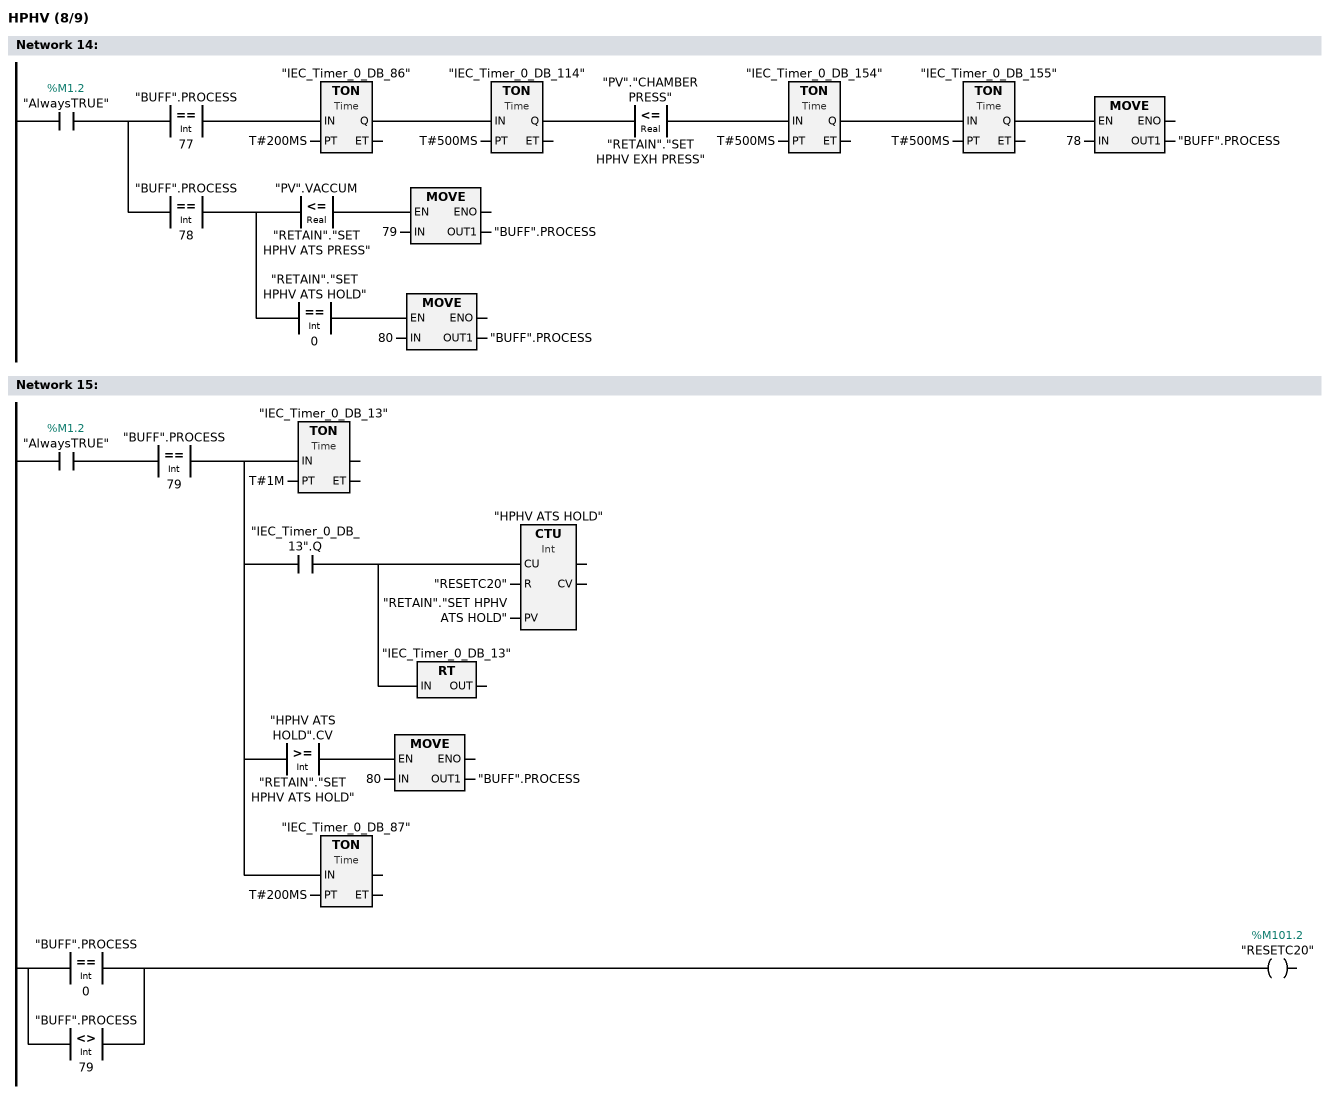
   RUNG wire#powerrail
      Contact( "AlwaysTRUE" )
      wire#w1
      { S7_Templates := "SrcType := Int" } EQ_Contact(in1 := "BUFF".PROCESS, in2 := 77)
      { S7_Templates := "time_type := Time" } "IEC_Timer_0_DB_86".TON(pt := T#200MS, et =>)
      { S7_Templates := "time_type := Time" } "IEC_Timer_0_DB_114".TON(pt := T#500MS, et =>)
      { S7_Templates := "SrcType := Real" } LE_Contact(in1 := "PV"."CHAMBER PRESS", in2 := "RETAIN"."SET HPHV EXH PRESS")
      { S7_Templates := "time_type := Time" } "IEC_Timer_0_DB_154".TON(pt := T#500MS, et =>)
      { S7_Templates := "time_type := Time" } "IEC_Timer_0_DB_155".TON(pt := T#500MS, et =>)
      Move(in := 78, out1 => "BUFF".PROCESS)
   END_RUNG
   RUNG wire#w1
      { S7_Templates := "SrcType := Int" } EQ_Contact(in1 := "BUFF".PROCESS, in2 := 78)
      wire#w2
      { S7_Templates := "SrcType := Real" } LE_Contact(in1 := "PV".VACCUM, in2 := "RETAIN"."SET HPHV ATS PRESS")
      Move(in := 79, out1 => "BUFF".PROCESS)
   END_RUNG
   RUNG wire#w2
      { S7_Templates := "SrcType := Int" } EQ_Contact(in1 := "RETAIN"."SET HPHV ATS HOLD", in2 := 0)
      Move(in := 80, out1 => "BUFF".PROCESS)
   END_RUNG
   // the same network as SCL:
   "IEC_Timer_0_DB_86".TON(IN := "AlwaysTRUE" AND ("BUFF".PROCESS = 77), PT := T#200MS);
   "IEC_Timer_0_DB_114".TON(IN := "IEC_Timer_0_DB_86".Q, PT := T#500MS);
   "IEC_Timer_0_DB_154".TON(IN := "IEC_Timer_0_DB_114".Q AND ("PV"."CHAMBER PRESS" <= "RETAIN"."SET HPHV EXH PRESS"),
                           PT := T#500MS);
   "IEC_Timer_0_DB_155".TON(IN := "IEC_Timer_0_DB_154".Q, PT := T#500MS);
   IF "IEC_Timer_0_DB_155".Q THEN "BUFF".PROCESS := 78; END_IF;
   #_w1 := "AlwaysTRUE" AND ("BUFF".PROCESS = 78);
   IF #_w1 AND ("PV".VACCUM <= "RETAIN"."SET HPHV ATS PRESS") THEN "BUFF".PROCESS := 79; END_IF;
   IF #_w1 AND ("RETAIN"."SET HPHV ATS HOLD" = 0) THEN "BUFF".PROCESS := 80; END_IF;
END_REGION

REGION Network 15
   RUNG wire#powerrail
      Contact( "AlwaysTRUE" )
      { S7_Templates := "SrcType := Int" } EQ_Contact(in1 := "BUFF".PROCESS, in2 := 79)
      wire#w1
      { S7_Templates := "time_type := Time" } "IEC_Timer_0_DB_13".TON(pt := T#1M, et =>)
   END_RUNG
   RUNG wire#w1
      Contact( "IEC_Timer_0_DB_13".Q )
      wire#w2
      { S7_Templates := "value_type := Int" } "HPHV ATS HOLD".CTU(r := "RESETC20", pv := "RETAIN"."SET HPHV ATS HOLD", cv =>)
   END_RUNG
   RUNG wire#w2
      RT_Coil( "IEC_Timer_0_DB_13" )
   END_RUNG
   RUNG wire#w1
      { S7_Templates := "SrcType := Int" } GE_Contact(in1 := "HPHV ATS HOLD".CV, in2 := "RETAIN"."SET HPHV ATS HOLD")
      Move(in := 80, out1 => "BUFF".PROCESS)
   END_RUNG
   RUNG wire#w1
      { S7_Templates := "time_type := Time" } "IEC_Timer_0_DB_87".TON(pt := T#200MS, et =>)
   END_RUNG
   RUNG wire#powerrail
      { S7_Templates := "SrcType := Int" } EQ_Contact(in1 := "BUFF".PROCESS, in2 := 0)
      wire#w3
      Coil( "RESETC20" )
   END_RUNG
   RUNG wire#powerrail
      { S7_Templates := "SrcType := Int" } NE_Contact(in1 := "BUFF".PROCESS, in2 := 79)
   END_RUNG wire#w3
   // the same network as SCL:
   #_w1 := "AlwaysTRUE" AND ("BUFF".PROCESS = 79);
   "IEC_Timer_0_DB_13".TON(IN := #_w1, PT := T#1M);
   #_w2 := #_w1 AND "IEC_Timer_0_DB_13".Q;
   "HPHV ATS HOLD".CTU(CU := #_w2, R := "RESETC20", PV := "RETAIN"."SET HPHV ATS HOLD");
   IF #_w2 THEN RESET_TIMER("IEC_Timer_0_DB_13"); END_IF;
   IF #_w1 AND ("HPHV ATS HOLD".CV >= "RETAIN"."SET HPHV ATS HOLD") THEN "BUFF".PROCESS := 80; END_IF;
   "IEC_Timer_0_DB_87".TON(IN := #_w1, PT := T#200MS);
   "RESETC20" := ("BUFF".PROCESS = 0) OR ("BUFF".PROCESS <> 79);
END_REGION

REGION Network 16
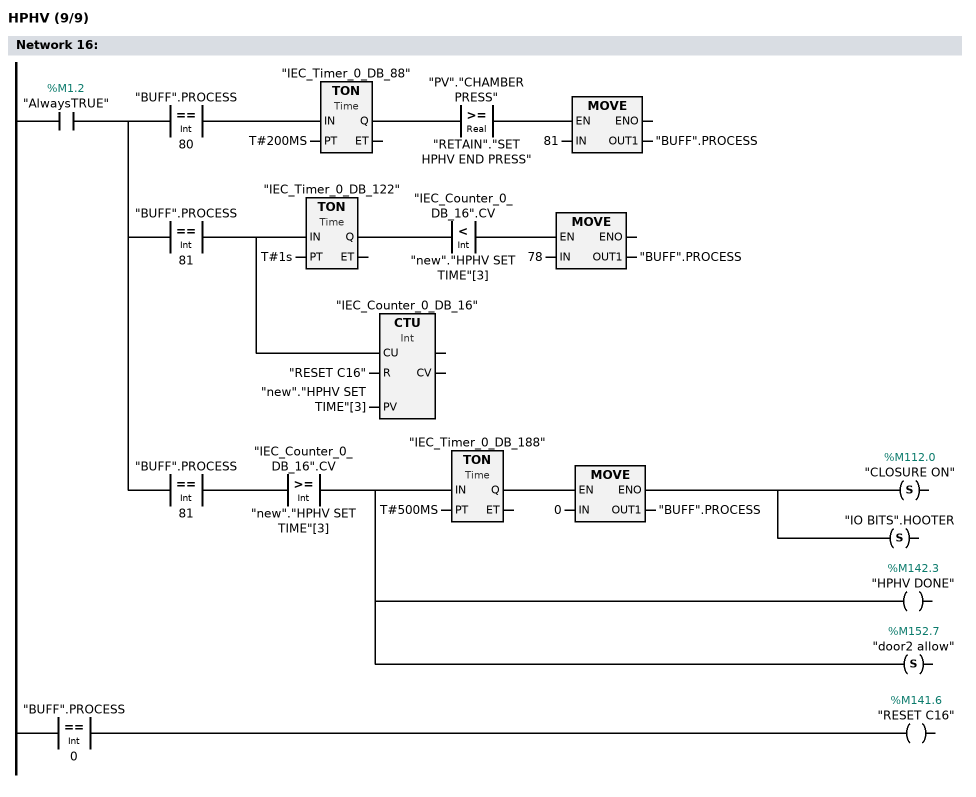
   RUNG wire#powerrail
      Contact( "AlwaysTRUE" )
      wire#w1
      { S7_Templates := "SrcType := Int" } EQ_Contact(in1 := "BUFF".PROCESS, in2 := 80)
      { S7_Templates := "time_type := Time" } "IEC_Timer_0_DB_88".TON(pt := T#200MS, et =>)
      { S7_Templates := "SrcType := Real" } GE_Contact(in1 := "PV"."CHAMBER PRESS", in2 := "RETAIN"."SET HPHV END PRESS")
      Move(in := 81, out1 => "BUFF".PROCESS)
   END_RUNG
   RUNG wire#w1
      { S7_Templates := "SrcType := Int" } EQ_Contact(in1 := "BUFF".PROCESS, in2 := 81)
      wire#w2
      { S7_Templates := "time_type := Time" } "IEC_Timer_0_DB_122".TON(pt := T#1s, et =>)
      { S7_Templates := "SrcType := Int" } LT_Contact(in1 := "IEC_Counter_0_DB_16".CV, in2 := "new"."HPHV SET TIME"[3])
      Move(in := 78, out1 => "BUFF".PROCESS)
   END_RUNG
   RUNG wire#w2
      { S7_Templates := "value_type := Int" } "IEC_Counter_0_DB_16".CTU(r := "RESET C16", pv := "new"."HPHV SET TIME"[3], cv =>)
   END_RUNG
   RUNG wire#w1
      { S7_Templates := "SrcType := Int" } EQ_Contact(in1 := "BUFF".PROCESS, in2 := 81)
      { S7_Templates := "SrcType := Int" } GE_Contact(in1 := "IEC_Counter_0_DB_16".CV, in2 := "new"."HPHV SET TIME"[3])
      wire#w3
      { S7_Templates := "time_type := Time" } "IEC_Timer_0_DB_188".TON(pt := T#500MS, et =>)
      Move(in := 0, out1 => "BUFF".PROCESS)
      wire#w4
      S_Coil( "CLOSURE ON" )
   END_RUNG
   RUNG wire#w4
      S_Coil( "IO BITS".HOOTER )
   END_RUNG
   RUNG wire#w3
      Coil( "HPHV DONE" )
   END_RUNG
   RUNG wire#w3
      S_Coil( "door2 allow" )
   END_RUNG
   RUNG wire#powerrail
      { S7_Templates := "SrcType := Int" } EQ_Contact(in1 := "BUFF".PROCESS, in2 := 0)
      Coil( "RESET C16" )
   END_RUNG
   // the same network as SCL:
   "IEC_Timer_0_DB_88".TON(IN := "AlwaysTRUE" AND ("BUFF".PROCESS = 80), PT := T#200MS);
   IF "IEC_Timer_0_DB_88".Q AND ("PV"."CHAMBER PRESS" >= "RETAIN"."SET HPHV END PRESS") THEN
       "BUFF".PROCESS := 81;
   END_IF;
   #_w1 := "AlwaysTRUE" AND ("BUFF".PROCESS = 81);
   "IEC_Timer_0_DB_122".TON(IN := #_w1, PT := T#1s);
   IF "IEC_Timer_0_DB_122".Q AND ("IEC_Counter_0_DB_16".CV < "new"."HPHV SET TIME"[3]) THEN
       "BUFF".PROCESS := 78;
   END_IF;
   "IEC_Counter_0_DB_16".CTU(CU := #_w1, R := "RESET C16", PV := "new"."HPHV SET TIME"[3]);
   #_w2 := "AlwaysTRUE" AND ("BUFF".PROCESS = 81) AND ("IEC_Counter_0_DB_16".CV >= "new"."HPHV SET TIME"[3]);
   "IEC_Timer_0_DB_188".TON(IN := #_w2, PT := T#500MS);
   IF "IEC_Timer_0_DB_188".Q THEN
       "BUFF".PROCESS := 0;
       "CLOSURE ON" := TRUE;
       "IO BITS".HOOTER := TRUE;
   END_IF;
   "HPHV DONE" := #_w2;
   IF #_w2 THEN "door2 allow" := TRUE; END_IF;
   "RESET C16" := "BUFF".PROCESS = 0;
END_REGION
END_FUNCTION

FUNCTION "BOWIE" : Void   // FC7, LAD
{ S7_Optimized_Access := 'TRUE' }
// stored: SetENOAutomatically false
   VAR_TEMP
      START : Bool;
   END_VAR
   VAR_TEMP   // added for the SCL form of the ladder/FBD networks
      _w1 : Bool;
      _w2 : Bool;
      _w3 : Bool;
      _w4 : Bool;
   END_VAR
BEGIN

REGION Network 1
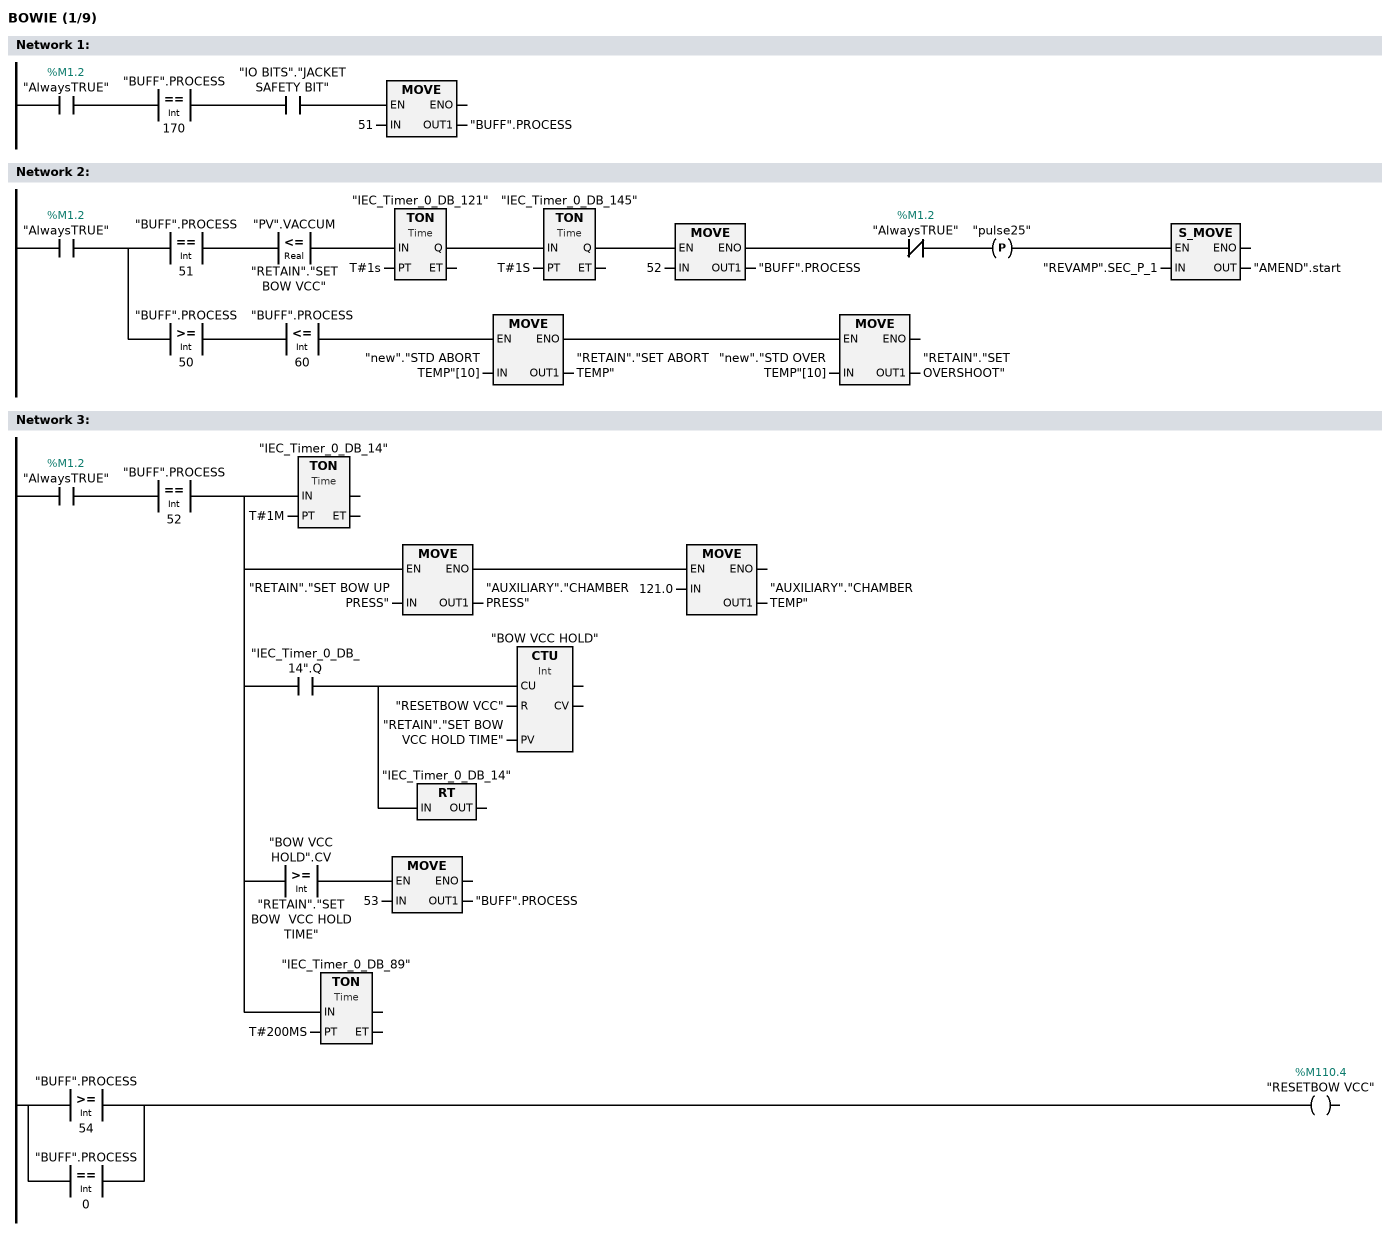
   RUNG wire#powerrail
      Contact( "AlwaysTRUE" )
      { S7_Templates := "SrcType := Int" } EQ_Contact(in1 := "BUFF".PROCESS, in2 := 170)
      Contact( "IO BITS"."JACKET SAFETY BIT" )
      Move(in := 51, out1 => "BUFF".PROCESS)
   END_RUNG
   // the same network as SCL:
   IF "AlwaysTRUE" AND ("BUFF".PROCESS = 170) AND "IO BITS"."JACKET SAFETY BIT" THEN
       "BUFF".PROCESS := 51;
   END_IF;
END_REGION

REGION Network 2
   RUNG wire#powerrail
      Contact( "AlwaysTRUE" )
      wire#w1
      { S7_Templates := "SrcType := Int" } EQ_Contact(in1 := "BUFF".PROCESS, in2 := 51)
      { S7_Templates := "SrcType := Real" } LE_Contact(in1 := "PV".VACCUM, in2 := "RETAIN"."SET BOW VCC")
      { S7_Templates := "time_type := Time" } "IEC_Timer_0_DB_121".TON(pt := T#1s, et =>)
      { S7_Templates := "time_type := Time" } "IEC_Timer_0_DB_145".TON(pt := T#1S, et =>)
      Move(in := 52, out1 => "BUFF".PROCESS)
      I_Contact( "AlwaysTRUE" )
      P_Trig( "pulse25" )
      S_Move(in := "REVAMP".SEC_P_1, out => "AMEND".start)
   END_RUNG
   RUNG wire#w1
      { S7_Templates := "SrcType := Int" } GE_Contact(in1 := "BUFF".PROCESS, in2 := 50)
      { S7_Templates := "SrcType := Int" } LE_Contact(in1 := "BUFF".PROCESS, in2 := 60)
      Move(in := "new"."STD ABORT TEMP"[10], out1 => "RETAIN"."SET ABORT TEMP")
      Move(in := "new"."STD OVER TEMP"[10], out1 => "RETAIN"."SET OVERSHOOT")
   END_RUNG
   // the same network as SCL:
   "IEC_Timer_0_DB_121".TON(IN := "AlwaysTRUE" AND ("BUFF".PROCESS = 51) AND ("PV".VACCUM <= "RETAIN"."SET BOW VCC"),
                           PT := T#1s);
   "IEC_Timer_0_DB_145".TON(IN := "IEC_Timer_0_DB_121".Q, PT := T#1S);
   IF "IEC_Timer_0_DB_145".Q THEN "BUFF".PROCESS := 52; END_IF;
   #_w1 := "IEC_Timer_0_DB_145".Q AND NOT "AlwaysTRUE";
   #_w2 := #_w1 AND NOT "pulse25";   // rising edge
   "pulse25" := #_w1;
   IF #_w2 THEN "AMEND".start := "REVAMP".SEC_P_1; END_IF;
   IF "AlwaysTRUE" AND ("BUFF".PROCESS >= 50) AND ("BUFF".PROCESS <= 60) THEN
       "RETAIN"."SET ABORT TEMP" := "new"."STD ABORT TEMP"[10];
       "RETAIN"."SET OVERSHOOT" := "new"."STD OVER TEMP"[10];
   END_IF;
END_REGION

REGION Network 3
   RUNG wire#powerrail
      Contact( "AlwaysTRUE" )
      { S7_Templates := "SrcType := Int" } EQ_Contact(in1 := "BUFF".PROCESS, in2 := 52)
      wire#w1
      { S7_Templates := "time_type := Time" } "IEC_Timer_0_DB_14".TON(pt := T#1M, et =>)
   END_RUNG
   RUNG wire#w1
      Move(in := "RETAIN"."SET BOW UP PRESS", out1 => "AUXILIARY"."CHAMBER PRESS")
      Move(in := 121.0, out1 => "AUXILIARY"."CHAMBER TEMP")
   END_RUNG
   RUNG wire#w1
      Contact( "IEC_Timer_0_DB_14".Q )
      wire#w2
      { S7_Templates := "value_type := Int" } "BOW VCC HOLD".CTU(r := "RESETBOW VCC", pv := "RETAIN"."SET BOW  VCC HOLD TIME", cv =>)
   END_RUNG
   RUNG wire#w2
      RT_Coil( "IEC_Timer_0_DB_14" )
   END_RUNG
   RUNG wire#w1
      { S7_Templates := "SrcType := Int" } GE_Contact(in1 := "BOW VCC HOLD".CV, in2 := "RETAIN"."SET BOW  VCC HOLD TIME")
      Move(in := 53, out1 => "BUFF".PROCESS)
   END_RUNG
   RUNG wire#w1
      { S7_Templates := "time_type := Time" } "IEC_Timer_0_DB_89".TON(pt := T#200MS, et =>)
   END_RUNG
   RUNG wire#powerrail
      { S7_Templates := "SrcType := Int" } GE_Contact(in1 := "BUFF".PROCESS, in2 := 54)
      wire#w3
      Coil( "RESETBOW VCC" )
   END_RUNG
   RUNG wire#powerrail
      { S7_Templates := "SrcType := Int" } EQ_Contact(in1 := "BUFF".PROCESS, in2 := 0)
   END_RUNG wire#w3
   // the same network as SCL:
   #_w1 := "AlwaysTRUE" AND ("BUFF".PROCESS = 52);
   "IEC_Timer_0_DB_14".TON(IN := #_w1, PT := T#1M);
   IF #_w1 THEN
       "AUXILIARY"."CHAMBER PRESS" := "RETAIN"."SET BOW UP PRESS";
       "AUXILIARY"."CHAMBER TEMP" := 121.0;
   END_IF;
   #_w2 := #_w1 AND "IEC_Timer_0_DB_14".Q;
   "BOW VCC HOLD".CTU(CU := #_w2, R := "RESETBOW VCC", PV := "RETAIN"."SET BOW  VCC HOLD TIME");
   IF #_w2 THEN RESET_TIMER("IEC_Timer_0_DB_14"); END_IF;
   IF #_w1 AND ("BOW VCC HOLD".CV >= "RETAIN"."SET BOW  VCC HOLD TIME") THEN "BUFF".PROCESS := 53; END_IF;
   "IEC_Timer_0_DB_89".TON(IN := #_w1, PT := T#200MS);
   "RESETBOW VCC" := ("BUFF".PROCESS >= 54) OR ("BUFF".PROCESS = 0);
END_REGION

REGION Network 4
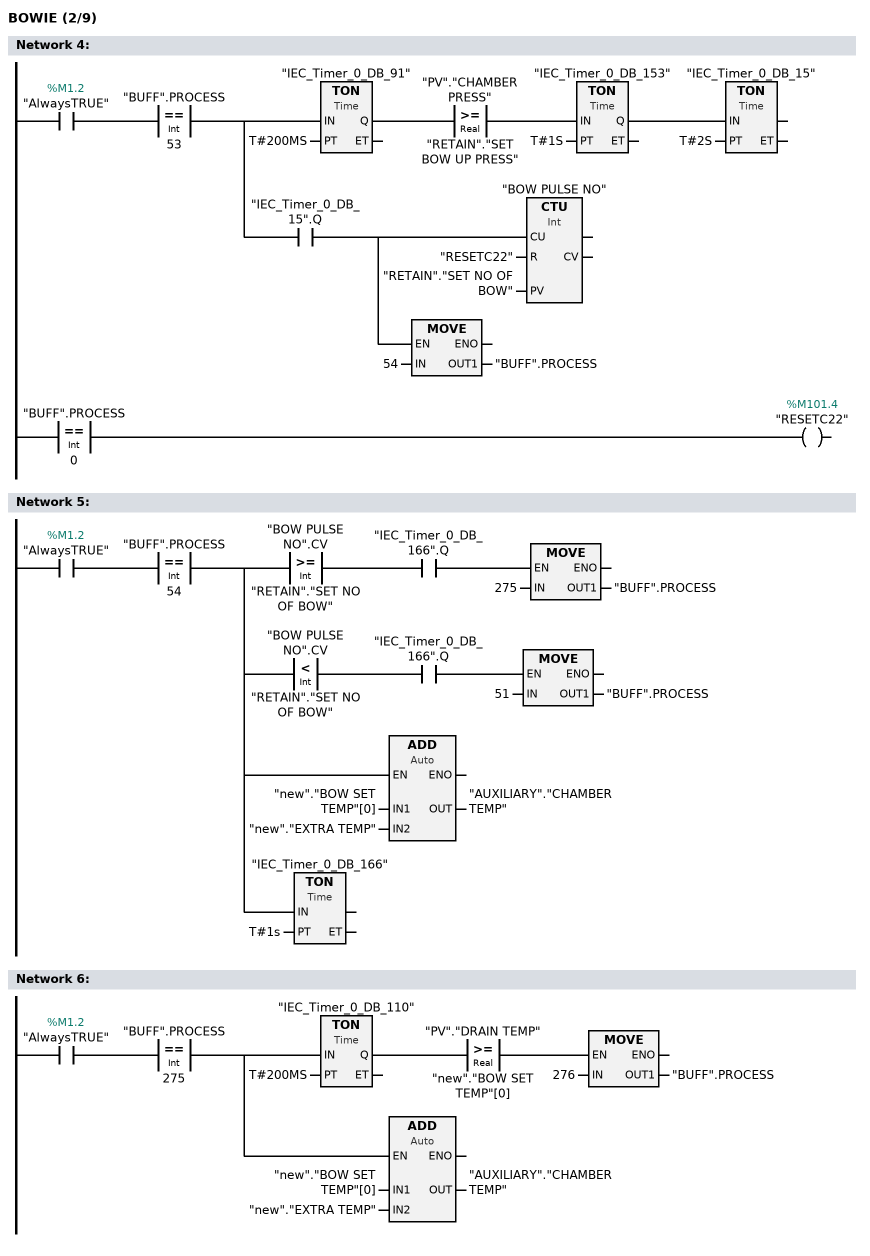
   RUNG wire#powerrail
      Contact( "AlwaysTRUE" )
      { S7_Templates := "SrcType := Int" } EQ_Contact(in1 := "BUFF".PROCESS, in2 := 53)
      wire#w1
      { S7_Templates := "time_type := Time" } "IEC_Timer_0_DB_91".TON(pt := T#200MS, et =>)
      { S7_Templates := "SrcType := Real" } GE_Contact(in1 := "PV"."CHAMBER PRESS", in2 := "RETAIN"."SET BOW UP PRESS")
      { S7_Templates := "time_type := Time" } "IEC_Timer_0_DB_153".TON(pt := T#1S, et =>)
      { S7_Templates := "time_type := Time" } "IEC_Timer_0_DB_15".TON(pt := T#2S, et =>)
   END_RUNG
   RUNG wire#w1
      Contact( "IEC_Timer_0_DB_15".Q )
      wire#w2
      { S7_Templates := "value_type := Int" } "BOW PULSE NO".CTU(r := "RESETC22", pv := "RETAIN"."SET NO OF BOW", cv =>)
   END_RUNG
   RUNG wire#w2
      Move(in := 54, out1 => "BUFF".PROCESS)
   END_RUNG
   RUNG wire#powerrail
      { S7_Templates := "SrcType := Int" } EQ_Contact(in1 := "BUFF".PROCESS, in2 := 0)
      Coil( "RESETC22" )
   END_RUNG
   // the same network as SCL:
   #_w1 := "AlwaysTRUE" AND ("BUFF".PROCESS = 53);
   "IEC_Timer_0_DB_91".TON(IN := #_w1, PT := T#200MS);
   "IEC_Timer_0_DB_153".TON(IN := "IEC_Timer_0_DB_91".Q AND ("PV"."CHAMBER PRESS" >= "RETAIN"."SET BOW UP PRESS"),
                           PT := T#1S);
   "IEC_Timer_0_DB_15".TON(IN := "IEC_Timer_0_DB_153".Q, PT := T#2S);
   #_w2 := #_w1 AND "IEC_Timer_0_DB_15".Q;
   "BOW PULSE NO".CTU(CU := #_w2, R := "RESETC22", PV := "RETAIN"."SET NO OF BOW");
   IF #_w2 THEN "BUFF".PROCESS := 54; END_IF;
   "RESETC22" := "BUFF".PROCESS = 0;
END_REGION

REGION Network 5
   RUNG wire#powerrail
      Contact( "AlwaysTRUE" )
      { S7_Templates := "SrcType := Int" } EQ_Contact(in1 := "BUFF".PROCESS, in2 := 54)
      wire#w1
      { S7_Templates := "SrcType := Int" } GE_Contact(in1 := "BOW PULSE NO".CV, in2 := "RETAIN"."SET NO OF BOW")
      Contact( "IEC_Timer_0_DB_166".Q )
      Move(in := 275, out1 => "BUFF".PROCESS)
   END_RUNG
   RUNG wire#w1
      { S7_Templates := "SrcType := Int" } LT_Contact(in1 := "BOW PULSE NO".CV, in2 := "RETAIN"."SET NO OF BOW")
      Contact( "IEC_Timer_0_DB_166".Q )
      Move(in := 51, out1 => "BUFF".PROCESS)
   END_RUNG
   RUNG wire#w1
      Add(in1 := "new"."BOW SET TEMP"[0], in2 := "new"."EXTRA TEMP", out => "AUXILIARY"."CHAMBER TEMP")
   END_RUNG
   RUNG wire#w1
      { S7_Templates := "time_type := Time" } "IEC_Timer_0_DB_166".TON(pt := T#1s, et =>)
   END_RUNG
   // the same network as SCL:
   #_w1 := "AlwaysTRUE" AND ("BUFF".PROCESS = 54);
   IF #_w1 AND ("BOW PULSE NO".CV >= "RETAIN"."SET NO OF BOW") AND "IEC_Timer_0_DB_166".Q THEN
       "BUFF".PROCESS := 275;
   END_IF;
   IF #_w1 AND ("BOW PULSE NO".CV < "RETAIN"."SET NO OF BOW") AND "IEC_Timer_0_DB_166".Q THEN
       "BUFF".PROCESS := 51;
   END_IF;
   IF #_w1 THEN "AUXILIARY"."CHAMBER TEMP" := "new"."BOW SET TEMP"[0] + "new"."EXTRA TEMP"; END_IF;
   "IEC_Timer_0_DB_166".TON(IN := #_w1, PT := T#1s);
END_REGION

REGION Network 6
   RUNG wire#powerrail
      Contact( "AlwaysTRUE" )
      { S7_Templates := "SrcType := Int" } EQ_Contact(in1 := "BUFF".PROCESS, in2 := 275)
      wire#w1
      { S7_Templates := "time_type := Time" } "IEC_Timer_0_DB_110".TON(pt := T#200MS, et =>)
      { S7_Templates := "SrcType := Real" } GE_Contact(in1 := "PV"."DRAIN TEMP", in2 := "new"."BOW SET TEMP"[0])
      Move(in := 276, out1 => "BUFF".PROCESS)
   END_RUNG
   RUNG wire#w1
      Add(in1 := "new"."BOW SET TEMP"[0], in2 := "new"."EXTRA TEMP", out => "AUXILIARY"."CHAMBER TEMP")
   END_RUNG
   // the same network as SCL:
   #_w1 := "AlwaysTRUE" AND ("BUFF".PROCESS = 275);
   "IEC_Timer_0_DB_110".TON(IN := #_w1, PT := T#200MS);
   IF "IEC_Timer_0_DB_110".Q AND ("PV"."DRAIN TEMP" >= "new"."BOW SET TEMP"[0]) THEN
       "BUFF".PROCESS := 276;
   END_IF;
   IF #_w1 THEN "AUXILIARY"."CHAMBER TEMP" := "new"."BOW SET TEMP"[0] + "new"."EXTRA TEMP"; END_IF;
END_REGION

REGION Network 7
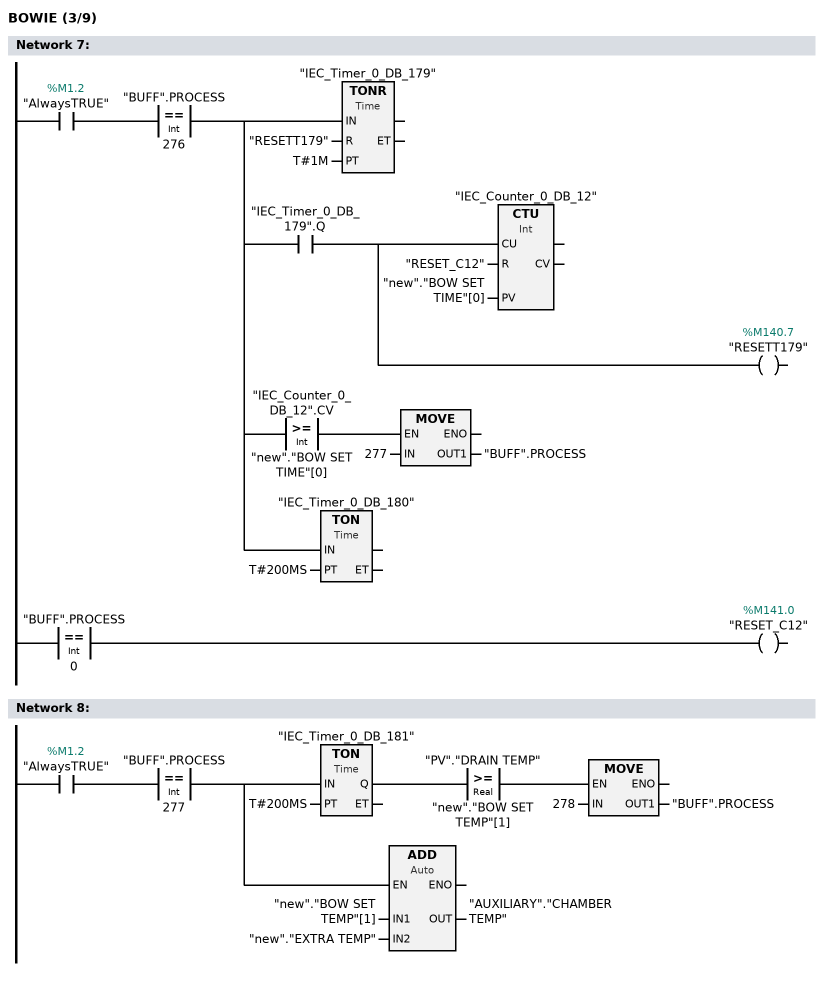
   RUNG wire#powerrail
      Contact( "AlwaysTRUE" )
      { S7_Templates := "SrcType := Int" } EQ_Contact(in1 := "BUFF".PROCESS, in2 := 276)
      wire#w1
      { S7_Templates := "time_type := Time" } "IEC_Timer_0_DB_179".TONR(r := "RESETT179", pt := T#1M, et =>)
   END_RUNG
   RUNG wire#w1
      Contact( "IEC_Timer_0_DB_179".Q )
      wire#w2
      { S7_Templates := "value_type := Int" } "IEC_Counter_0_DB_12".CTU(r := "RESET_C12", pv := "new"."BOW SET TIME"[0], cv =>)
   END_RUNG
   RUNG wire#w2
      Coil( "RESETT179" )
   END_RUNG
   RUNG wire#w1
      { S7_Templates := "SrcType := Int" } GE_Contact(in1 := "IEC_Counter_0_DB_12".CV, in2 := "new"."BOW SET TIME"[0])
      Move(in := 277, out1 => "BUFF".PROCESS)
   END_RUNG
   RUNG wire#w1
      { S7_Templates := "time_type := Time" } "IEC_Timer_0_DB_180".TON(pt := T#200MS, et =>)
   END_RUNG
   RUNG wire#powerrail
      { S7_Templates := "SrcType := Int" } EQ_Contact(in1 := "BUFF".PROCESS, in2 := 0)
      Coil( "RESET_C12" )
   END_RUNG
   // the same network as SCL:
   #_w1 := "AlwaysTRUE" AND ("BUFF".PROCESS = 276);
   "IEC_Timer_0_DB_179".TONR(IN := #_w1, R := "RESETT179", PT := T#1M);
   #_w2 := #_w1 AND "IEC_Timer_0_DB_179".Q;
   "IEC_Counter_0_DB_12".CTU(CU := #_w2, R := "RESET_C12", PV := "new"."BOW SET TIME"[0]);
   "RESETT179" := #_w2;
   IF #_w1 AND ("IEC_Counter_0_DB_12".CV >= "new"."BOW SET TIME"[0]) THEN "BUFF".PROCESS := 277; END_IF;
   "IEC_Timer_0_DB_180".TON(IN := #_w1, PT := T#200MS);
   "RESET_C12" := "BUFF".PROCESS = 0;
END_REGION

REGION Network 8
   RUNG wire#powerrail
      Contact( "AlwaysTRUE" )
      { S7_Templates := "SrcType := Int" } EQ_Contact(in1 := "BUFF".PROCESS, in2 := 277)
      wire#w1
      { S7_Templates := "time_type := Time" } "IEC_Timer_0_DB_181".TON(pt := T#200MS, et =>)
      { S7_Templates := "SrcType := Real" } GE_Contact(in1 := "PV"."DRAIN TEMP", in2 := "new"."BOW SET TEMP"[1])
      Move(in := 278, out1 => "BUFF".PROCESS)
   END_RUNG
   RUNG wire#w1
      Add(in1 := "new"."BOW SET TEMP"[1], in2 := "new"."EXTRA TEMP", out => "AUXILIARY"."CHAMBER TEMP")
   END_RUNG
   // the same network as SCL:
   #_w1 := "AlwaysTRUE" AND ("BUFF".PROCESS = 277);
   "IEC_Timer_0_DB_181".TON(IN := #_w1, PT := T#200MS);
   IF "IEC_Timer_0_DB_181".Q AND ("PV"."DRAIN TEMP" >= "new"."BOW SET TEMP"[1]) THEN
       "BUFF".PROCESS := 278;
   END_IF;
   IF #_w1 THEN "AUXILIARY"."CHAMBER TEMP" := "new"."BOW SET TEMP"[1] + "new"."EXTRA TEMP"; END_IF;
END_REGION

REGION Network 9
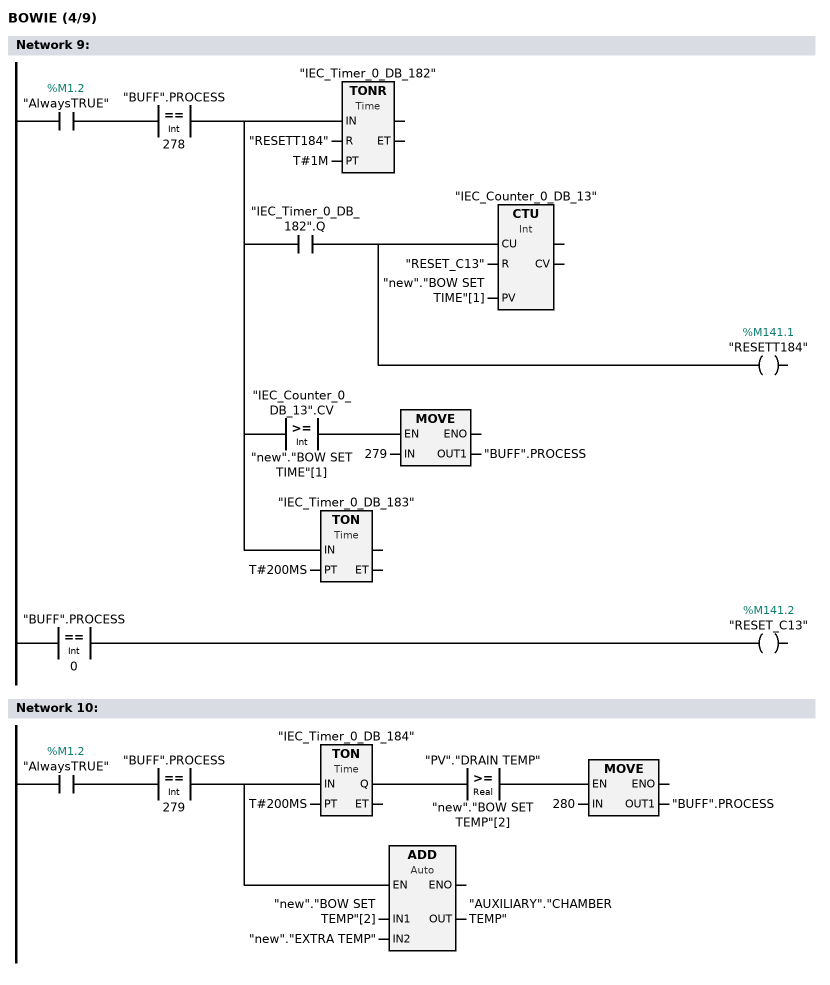
   RUNG wire#powerrail
      Contact( "AlwaysTRUE" )
      { S7_Templates := "SrcType := Int" } EQ_Contact(in1 := "BUFF".PROCESS, in2 := 278)
      wire#w1
      { S7_Templates := "time_type := Time" } "IEC_Timer_0_DB_182".TONR(r := "RESETT184", pt := T#1M, et =>)
   END_RUNG
   RUNG wire#w1
      Contact( "IEC_Timer_0_DB_182".Q )
      wire#w2
      { S7_Templates := "value_type := Int" } "IEC_Counter_0_DB_13".CTU(r := "RESET_C13", pv := "new"."BOW SET TIME"[1], cv =>)
   END_RUNG
   RUNG wire#w2
      Coil( "RESETT184" )
   END_RUNG
   RUNG wire#w1
      { S7_Templates := "SrcType := Int" } GE_Contact(in1 := "IEC_Counter_0_DB_13".CV, in2 := "new"."BOW SET TIME"[1])
      Move(in := 279, out1 => "BUFF".PROCESS)
   END_RUNG
   RUNG wire#w1
      { S7_Templates := "time_type := Time" } "IEC_Timer_0_DB_183".TON(pt := T#200MS, et =>)
   END_RUNG
   RUNG wire#powerrail
      { S7_Templates := "SrcType := Int" } EQ_Contact(in1 := "BUFF".PROCESS, in2 := 0)
      Coil( "RESET_C13" )
   END_RUNG
   // the same network as SCL:
   #_w1 := "AlwaysTRUE" AND ("BUFF".PROCESS = 278);
   "IEC_Timer_0_DB_182".TONR(IN := #_w1, R := "RESETT184", PT := T#1M);
   #_w2 := #_w1 AND "IEC_Timer_0_DB_182".Q;
   "IEC_Counter_0_DB_13".CTU(CU := #_w2, R := "RESET_C13", PV := "new"."BOW SET TIME"[1]);
   "RESETT184" := #_w2;
   IF #_w1 AND ("IEC_Counter_0_DB_13".CV >= "new"."BOW SET TIME"[1]) THEN "BUFF".PROCESS := 279; END_IF;
   "IEC_Timer_0_DB_183".TON(IN := #_w1, PT := T#200MS);
   "RESET_C13" := "BUFF".PROCESS = 0;
END_REGION

REGION Network 10
   RUNG wire#powerrail
      Contact( "AlwaysTRUE" )
      { S7_Templates := "SrcType := Int" } EQ_Contact(in1 := "BUFF".PROCESS, in2 := 279)
      wire#w1
      { S7_Templates := "time_type := Time" } "IEC_Timer_0_DB_184".TON(pt := T#200MS, et =>)
      { S7_Templates := "SrcType := Real" } GE_Contact(in1 := "PV"."DRAIN TEMP", in2 := "new"."BOW SET TEMP"[2])
      Move(in := 280, out1 => "BUFF".PROCESS)
   END_RUNG
   RUNG wire#w1
      Add(in1 := "new"."BOW SET TEMP"[2], in2 := "new"."EXTRA TEMP", out => "AUXILIARY"."CHAMBER TEMP")
   END_RUNG
   // the same network as SCL:
   #_w1 := "AlwaysTRUE" AND ("BUFF".PROCESS = 279);
   "IEC_Timer_0_DB_184".TON(IN := #_w1, PT := T#200MS);
   IF "IEC_Timer_0_DB_184".Q AND ("PV"."DRAIN TEMP" >= "new"."BOW SET TEMP"[2]) THEN
       "BUFF".PROCESS := 280;
   END_IF;
   IF #_w1 THEN "AUXILIARY"."CHAMBER TEMP" := "new"."BOW SET TEMP"[2] + "new"."EXTRA TEMP"; END_IF;
END_REGION

REGION Network 11
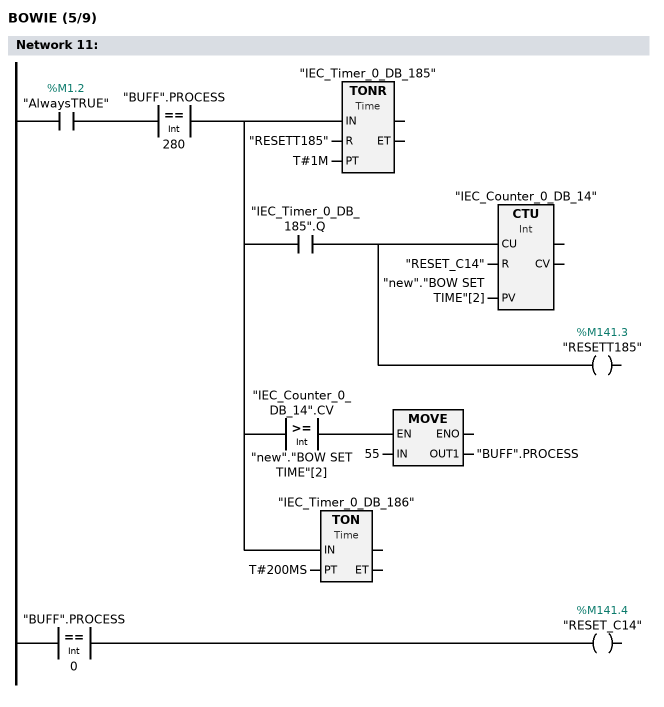
   RUNG wire#powerrail
      Contact( "AlwaysTRUE" )
      { S7_Templates := "SrcType := Int" } EQ_Contact(in1 := "BUFF".PROCESS, in2 := 280)
      wire#w1
      { S7_Templates := "time_type := Time" } "IEC_Timer_0_DB_185".TONR(r := "RESETT185", pt := T#1M, et =>)
   END_RUNG
   RUNG wire#w1
      Contact( "IEC_Timer_0_DB_185".Q )
      wire#w2
      { S7_Templates := "value_type := Int" } "IEC_Counter_0_DB_14".CTU(r := "RESET_C14", pv := "new"."BOW SET TIME"[2], cv =>)
   END_RUNG
   RUNG wire#w2
      Coil( "RESETT185" )
   END_RUNG
   RUNG wire#w1
      { S7_Templates := "SrcType := Int" } GE_Contact(in1 := "IEC_Counter_0_DB_14".CV, in2 := "new"."BOW SET TIME"[2])
      Move(in := 55, out1 => "BUFF".PROCESS)
   END_RUNG
   RUNG wire#w1
      { S7_Templates := "time_type := Time" } "IEC_Timer_0_DB_186".TON(pt := T#200MS, et =>)
   END_RUNG
   RUNG wire#powerrail
      { S7_Templates := "SrcType := Int" } EQ_Contact(in1 := "BUFF".PROCESS, in2 := 0)
      Coil( "RESET_C14" )
   END_RUNG
   // the same network as SCL:
   #_w1 := "AlwaysTRUE" AND ("BUFF".PROCESS = 280);
   "IEC_Timer_0_DB_185".TONR(IN := #_w1, R := "RESETT185", PT := T#1M);
   #_w2 := #_w1 AND "IEC_Timer_0_DB_185".Q;
   "IEC_Counter_0_DB_14".CTU(CU := #_w2, R := "RESET_C14", PV := "new"."BOW SET TIME"[2]);
   "RESETT185" := #_w2;
   IF #_w1 AND ("IEC_Counter_0_DB_14".CV >= "new"."BOW SET TIME"[2]) THEN "BUFF".PROCESS := 55; END_IF;
   "IEC_Timer_0_DB_186".TON(IN := #_w1, PT := T#200MS);
   "RESET_C14" := "BUFF".PROCESS = 0;
END_REGION

REGION Network 12
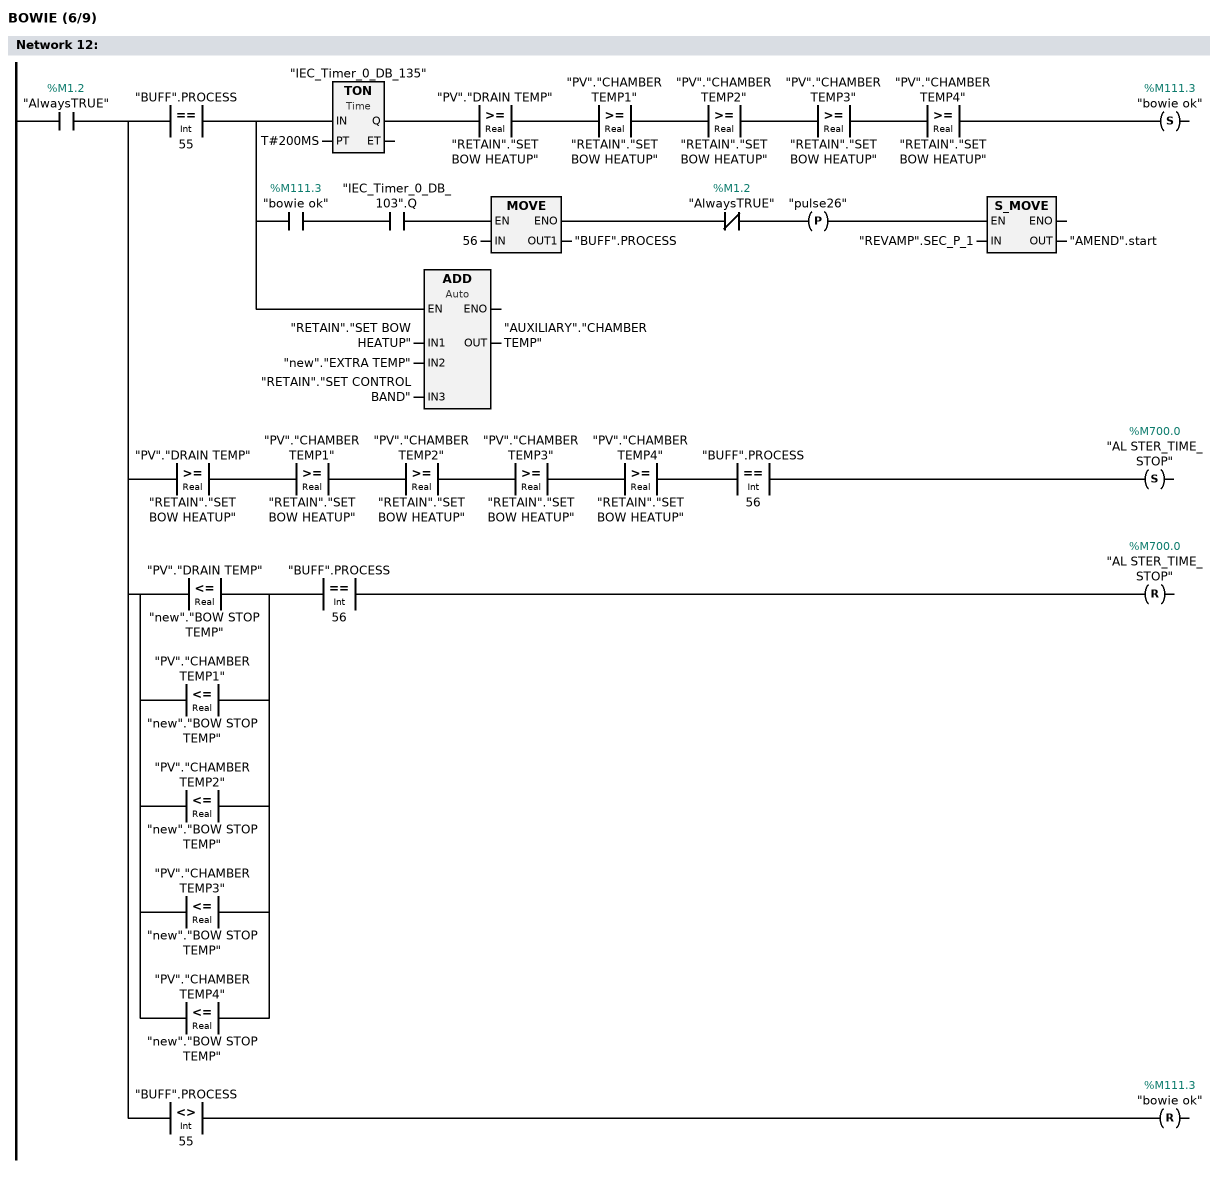
   RUNG wire#powerrail
      Contact( "AlwaysTRUE" )
      wire#w1
      { S7_Templates := "SrcType := Int" } EQ_Contact(in1 := "BUFF".PROCESS, in2 := 55)
      wire#w2
      { S7_Templates := "time_type := Time" } "IEC_Timer_0_DB_135".TON(pt := T#200MS, et =>)
      { S7_Templates := "SrcType := Real" } GE_Contact(in1 := "PV"."DRAIN TEMP", in2 := "RETAIN"."SET BOW HEATUP")
      { S7_Templates := "SrcType := Real" } GE_Contact(in1 := "PV"."CHAMBER TEMP1", in2 := "RETAIN"."SET BOW HEATUP")
      { S7_Templates := "SrcType := Real" } GE_Contact(in1 := "PV"."CHAMBER TEMP2", in2 := "RETAIN"."SET BOW HEATUP")
      { S7_Templates := "SrcType := Real" } GE_Contact(in1 := "PV"."CHAMBER TEMP3", in2 := "RETAIN"."SET BOW HEATUP")
      { S7_Templates := "SrcType := Real" } GE_Contact(in1 := "PV"."CHAMBER TEMP4", in2 := "RETAIN"."SET BOW HEATUP")
      S_Coil( "bowie ok" )
   END_RUNG
   RUNG wire#w2
      Contact( "bowie ok" )
      Contact( "IEC_Timer_0_DB_103".Q )
      Move(in := 56, out1 => "BUFF".PROCESS)
      I_Contact( "AlwaysTRUE" )
      P_Trig( "pulse26" )
      S_Move(in := "REVAMP".SEC_P_1, out => "AMEND".start)
   END_RUNG
   RUNG wire#w2
      Add(in1 := "RETAIN"."SET BOW HEATUP", in2 := "new"."EXTRA TEMP", in3 := "RETAIN"."SET CONTROL BAND", out => "AUXILIARY"."CHAMBER TEMP")
   END_RUNG
   RUNG wire#w1
      { S7_Templates := "SrcType := Real" } GE_Contact(in1 := "PV"."DRAIN TEMP", in2 := "RETAIN"."SET BOW HEATUP")
      { S7_Templates := "SrcType := Real" } GE_Contact(in1 := "PV"."CHAMBER TEMP1", in2 := "RETAIN"."SET BOW HEATUP")
      { S7_Templates := "SrcType := Real" } GE_Contact(in1 := "PV"."CHAMBER TEMP2", in2 := "RETAIN"."SET BOW HEATUP")
      { S7_Templates := "SrcType := Real" } GE_Contact(in1 := "PV"."CHAMBER TEMP3", in2 := "RETAIN"."SET BOW HEATUP")
      { S7_Templates := "SrcType := Real" } GE_Contact(in1 := "PV"."CHAMBER TEMP4", in2 := "RETAIN"."SET BOW HEATUP")
      { S7_Templates := "SrcType := Int" } EQ_Contact(in1 := "BUFF".PROCESS, in2 := 56)
      S_Coil( "AL STER_TIME_STOP" )
   END_RUNG
   RUNG wire#w1
      { S7_Templates := "SrcType := Real" } LE_Contact(in1 := "PV"."DRAIN TEMP", in2 := "new"."BOW STOP TEMP")
      wire#w3
      { S7_Templates := "SrcType := Int" } EQ_Contact(in1 := "BUFF".PROCESS, in2 := 56)
      R_Coil( "AL STER_TIME_STOP" )
   END_RUNG
   RUNG wire#w1
      { S7_Templates := "SrcType := Real" } LE_Contact(in1 := "PV"."CHAMBER TEMP1", in2 := "new"."BOW STOP TEMP")
   END_RUNG wire#w3
   RUNG wire#w1
      { S7_Templates := "SrcType := Real" } LE_Contact(in1 := "PV"."CHAMBER TEMP2", in2 := "new"."BOW STOP TEMP")
   END_RUNG wire#w3
   RUNG wire#w1
      { S7_Templates := "SrcType := Real" } LE_Contact(in1 := "PV"."CHAMBER TEMP3", in2 := "new"."BOW STOP TEMP")
   END_RUNG wire#w3
   RUNG wire#w1
      { S7_Templates := "SrcType := Real" } LE_Contact(in1 := "PV"."CHAMBER TEMP4", in2 := "new"."BOW STOP TEMP")
   END_RUNG wire#w3
   RUNG wire#w1
      { S7_Templates := "SrcType := Int" } NE_Contact(in1 := "BUFF".PROCESS, in2 := 55)
      R_Coil( "bowie ok" )
   END_RUNG
   // the same network as SCL:
   #_w1 := "AlwaysTRUE" AND ("BUFF".PROCESS = 55);
   "IEC_Timer_0_DB_135".TON(IN := #_w1, PT := T#200MS);
   IF "IEC_Timer_0_DB_135".Q AND ("PV"."DRAIN TEMP" >= "RETAIN"."SET BOW HEATUP") AND ("PV"."CHAMBER TEMP1" >= "RETAIN"."SET BOW HEATUP") AND ("PV"."CHAMBER TEMP2" >= "RETAIN"."SET BOW HEATUP") AND ("PV"."CHAMBER TEMP3" >= "RETAIN"."SET BOW HEATUP") AND ("PV"."CHAMBER TEMP4" >= "RETAIN"."SET BOW HEATUP") THEN
       "bowie ok" := TRUE;
   END_IF;
   #_w2 := #_w1 AND "bowie ok" AND "IEC_Timer_0_DB_103".Q;
   IF #_w2 THEN "BUFF".PROCESS := 56; END_IF;
   #_w3 := #_w2 AND NOT "AlwaysTRUE";
   #_w4 := #_w3 AND NOT "pulse26";   // rising edge
   "pulse26" := #_w3;
   IF #_w4 THEN "AMEND".start := "REVAMP".SEC_P_1; END_IF;
   IF #_w1 THEN
       "AUXILIARY"."CHAMBER TEMP" := "RETAIN"."SET BOW HEATUP" + "new"."EXTRA TEMP" + "RETAIN"."SET CONTROL BAND";
   END_IF;
   IF "AlwaysTRUE" AND ("PV"."DRAIN TEMP" >= "RETAIN"."SET BOW HEATUP") AND ("PV"."CHAMBER TEMP1" >= "RETAIN"."SET BOW HEATUP") AND ("PV"."CHAMBER TEMP2" >= "RETAIN"."SET BOW HEATUP") AND ("PV"."CHAMBER TEMP3" >= "RETAIN"."SET BOW HEATUP") AND ("PV"."CHAMBER TEMP4" >= "RETAIN"."SET BOW HEATUP") AND ("BUFF".PROCESS = 56) THEN
       "AL STER_TIME_STOP" := TRUE;
   END_IF;
   IF "AlwaysTRUE" AND (("PV"."DRAIN TEMP" <= "new"."BOW STOP TEMP") OR ("PV"."CHAMBER TEMP1" <= "new"."BOW STOP TEMP") OR ("PV"."CHAMBER TEMP2" <= "new"."BOW STOP TEMP") OR ("PV"."CHAMBER TEMP3" <= "new"."BOW STOP TEMP") OR ("PV"."CHAMBER TEMP4" <= "new"."BOW STOP TEMP")) AND ("BUFF".PROCESS = 56) THEN
       "AL STER_TIME_STOP" := FALSE;
   END_IF;
   IF "AlwaysTRUE" AND ("BUFF".PROCESS <> 55) THEN "bowie ok" := FALSE; END_IF;
END_REGION

REGION Network 13
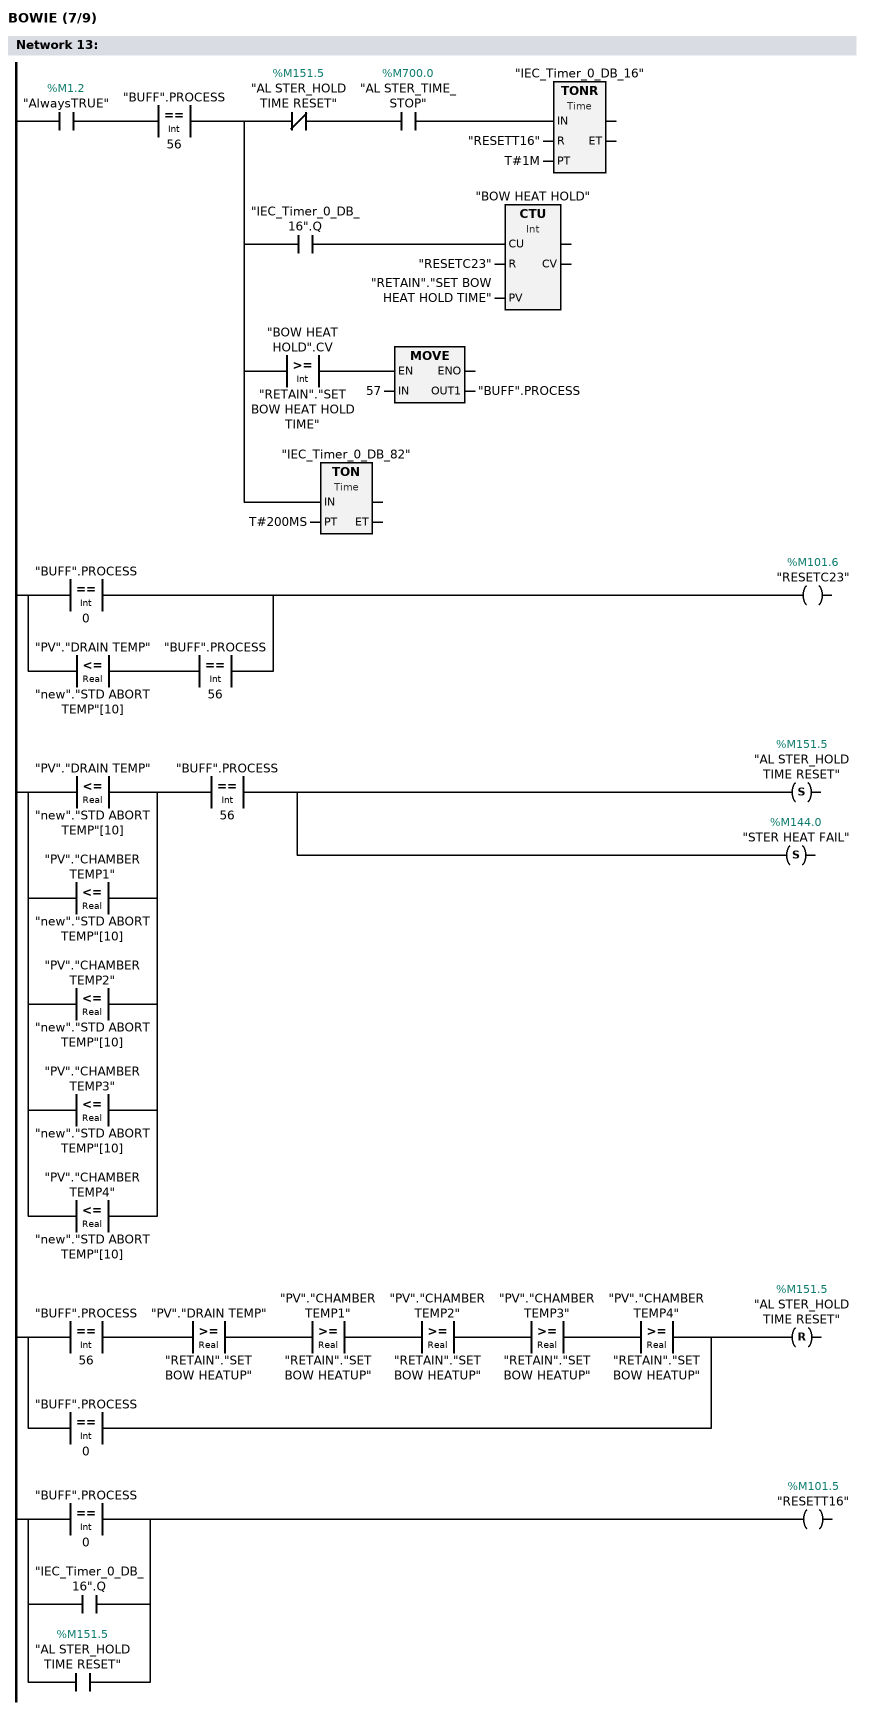
   RUNG wire#powerrail
      Contact( "AlwaysTRUE" )
      { S7_Templates := "SrcType := Int" } EQ_Contact(in1 := "BUFF".PROCESS, in2 := 56)
      wire#w1
      I_Contact( "AL STER_HOLD TIME RESET" )
      Contact( "AL STER_TIME_STOP" )
      { S7_Templates := "time_type := Time" } "IEC_Timer_0_DB_16".TONR(r := "RESETT16", pt := T#1M, et =>)
   END_RUNG
   RUNG wire#w1
      Contact( "IEC_Timer_0_DB_16".Q )
      { S7_Templates := "value_type := Int" } "BOW HEAT HOLD".CTU(r := "RESETC23", pv := "RETAIN"."SET BOW HEAT HOLD TIME", cv =>)
   END_RUNG
   RUNG wire#w1
      { S7_Templates := "SrcType := Int" } GE_Contact(in1 := "BOW HEAT HOLD".CV, in2 := "RETAIN"."SET BOW HEAT HOLD TIME")
      Move(in := 57, out1 => "BUFF".PROCESS)
   END_RUNG
   RUNG wire#w1
      { S7_Templates := "time_type := Time" } "IEC_Timer_0_DB_82".TON(pt := T#200MS, et =>)
   END_RUNG
   RUNG wire#powerrail
      { S7_Templates := "SrcType := Int" } EQ_Contact(in1 := "BUFF".PROCESS, in2 := 0)
      wire#w2
      Coil( "RESETC23" )
   END_RUNG
   RUNG wire#powerrail
      { S7_Templates := "SrcType := Real" } LE_Contact(in1 := "PV"."DRAIN TEMP", in2 := "new"."STD ABORT TEMP"[10])
      { S7_Templates := "SrcType := Int" } EQ_Contact(in1 := "BUFF".PROCESS, in2 := 56)
   END_RUNG wire#w2
   RUNG wire#powerrail
      { S7_Templates := "SrcType := Real" } LE_Contact(in1 := "PV"."DRAIN TEMP", in2 := "new"."STD ABORT TEMP"[10])
      wire#w3
      { S7_Templates := "SrcType := Int" } EQ_Contact(in1 := "BUFF".PROCESS, in2 := 56)
      wire#w4
      S_Coil( "AL STER_HOLD TIME RESET" )
   END_RUNG
   RUNG wire#powerrail
      { S7_Templates := "SrcType := Real" } LE_Contact(in1 := "PV"."CHAMBER TEMP1", in2 := "new"."STD ABORT TEMP"[10])
   END_RUNG wire#w3
   RUNG wire#powerrail
      { S7_Templates := "SrcType := Real" } LE_Contact(in1 := "PV"."CHAMBER TEMP2", in2 := "new"."STD ABORT TEMP"[10])
   END_RUNG wire#w3
   RUNG wire#powerrail
      { S7_Templates := "SrcType := Real" } LE_Contact(in1 := "PV"."CHAMBER TEMP3", in2 := "new"."STD ABORT TEMP"[10])
   END_RUNG wire#w3
   RUNG wire#powerrail
      { S7_Templates := "SrcType := Real" } LE_Contact(in1 := "PV"."CHAMBER TEMP4", in2 := "new"."STD ABORT TEMP"[10])
   END_RUNG wire#w3
   RUNG wire#w4
      S_Coil( "STER HEAT FAIL" )
   END_RUNG
   RUNG wire#powerrail
      { S7_Templates := "SrcType := Int" } EQ_Contact(in1 := "BUFF".PROCESS, in2 := 56)
      { S7_Templates := "SrcType := Real" } GE_Contact(in1 := "PV"."DRAIN TEMP", in2 := "RETAIN"."SET BOW HEATUP")
      { S7_Templates := "SrcType := Real" } GE_Contact(in1 := "PV"."CHAMBER TEMP1", in2 := "RETAIN"."SET BOW HEATUP")
      { S7_Templates := "SrcType := Real" } GE_Contact(in1 := "PV"."CHAMBER TEMP2", in2 := "RETAIN"."SET BOW HEATUP")
      { S7_Templates := "SrcType := Real" } GE_Contact(in1 := "PV"."CHAMBER TEMP3", in2 := "RETAIN"."SET BOW HEATUP")
      { S7_Templates := "SrcType := Real" } GE_Contact(in1 := "PV"."CHAMBER TEMP4", in2 := "RETAIN"."SET BOW HEATUP")
      wire#w5
      R_Coil( "AL STER_HOLD TIME RESET" )
   END_RUNG
   RUNG wire#powerrail
      { S7_Templates := "SrcType := Int" } EQ_Contact(in1 := "BUFF".PROCESS, in2 := 0)
   END_RUNG wire#w5
   RUNG wire#powerrail
      { S7_Templates := "SrcType := Int" } EQ_Contact(in1 := "BUFF".PROCESS, in2 := 0)
      wire#w6
      Coil( "RESETT16" )
   END_RUNG
   RUNG wire#powerrail
      Contact( "IEC_Timer_0_DB_16".Q )
   END_RUNG wire#w6
   RUNG wire#powerrail
      Contact( "AL STER_HOLD TIME RESET" )
   END_RUNG wire#w6
   // the same network as SCL:
   #_w1 := "AlwaysTRUE" AND ("BUFF".PROCESS = 56);
   "IEC_Timer_0_DB_16".TONR(IN := #_w1 AND NOT "AL STER_HOLD TIME RESET" AND "AL STER_TIME_STOP",
                           R := "RESETT16",
                           PT := T#1M);
   "BOW HEAT HOLD".CTU(CU := #_w1 AND "IEC_Timer_0_DB_16".Q,
                       R := "RESETC23",
                       PV := "RETAIN"."SET BOW HEAT HOLD TIME");
   IF #_w1 AND ("BOW HEAT HOLD".CV >= "RETAIN"."SET BOW HEAT HOLD TIME") THEN "BUFF".PROCESS := 57; END_IF;
   "IEC_Timer_0_DB_82".TON(IN := #_w1, PT := T#200MS);
   "RESETC23" := ("BUFF".PROCESS = 0) OR (("PV"."DRAIN TEMP" <= "new"."STD ABORT TEMP"[10]) AND ("BUFF".PROCESS = 56));
   IF (("PV"."DRAIN TEMP" <= "new"."STD ABORT TEMP"[10]) OR ("PV"."CHAMBER TEMP1" <= "new"."STD ABORT TEMP"[10]) OR ("PV"."CHAMBER TEMP2" <= "new"."STD ABORT TEMP"[10]) OR ("PV"."CHAMBER TEMP3" <= "new"."STD ABORT TEMP"[10]) OR ("PV"."CHAMBER TEMP4" <= "new"."STD ABORT TEMP"[10])) AND ("BUFF".PROCESS = 56) THEN
       "AL STER_HOLD TIME RESET" := TRUE;
       "STER HEAT FAIL" := TRUE;
   END_IF;
   IF (("BUFF".PROCESS = 56) AND ("PV"."DRAIN TEMP" >= "RETAIN"."SET BOW HEATUP") AND ("PV"."CHAMBER TEMP1" >= "RETAIN"."SET BOW HEATUP") AND ("PV"."CHAMBER TEMP2" >= "RETAIN"."SET BOW HEATUP") AND ("PV"."CHAMBER TEMP3" >= "RETAIN"."SET BOW HEATUP") AND ("PV"."CHAMBER TEMP4" >= "RETAIN"."SET BOW HEATUP")) OR ("BUFF".PROCESS = 0) THEN
       "AL STER_HOLD TIME RESET" := FALSE;
   END_IF;
   "RESETT16" := ("BUFF".PROCESS = 0) OR "IEC_Timer_0_DB_16".Q OR "AL STER_HOLD TIME RESET";
END_REGION

REGION Network 14
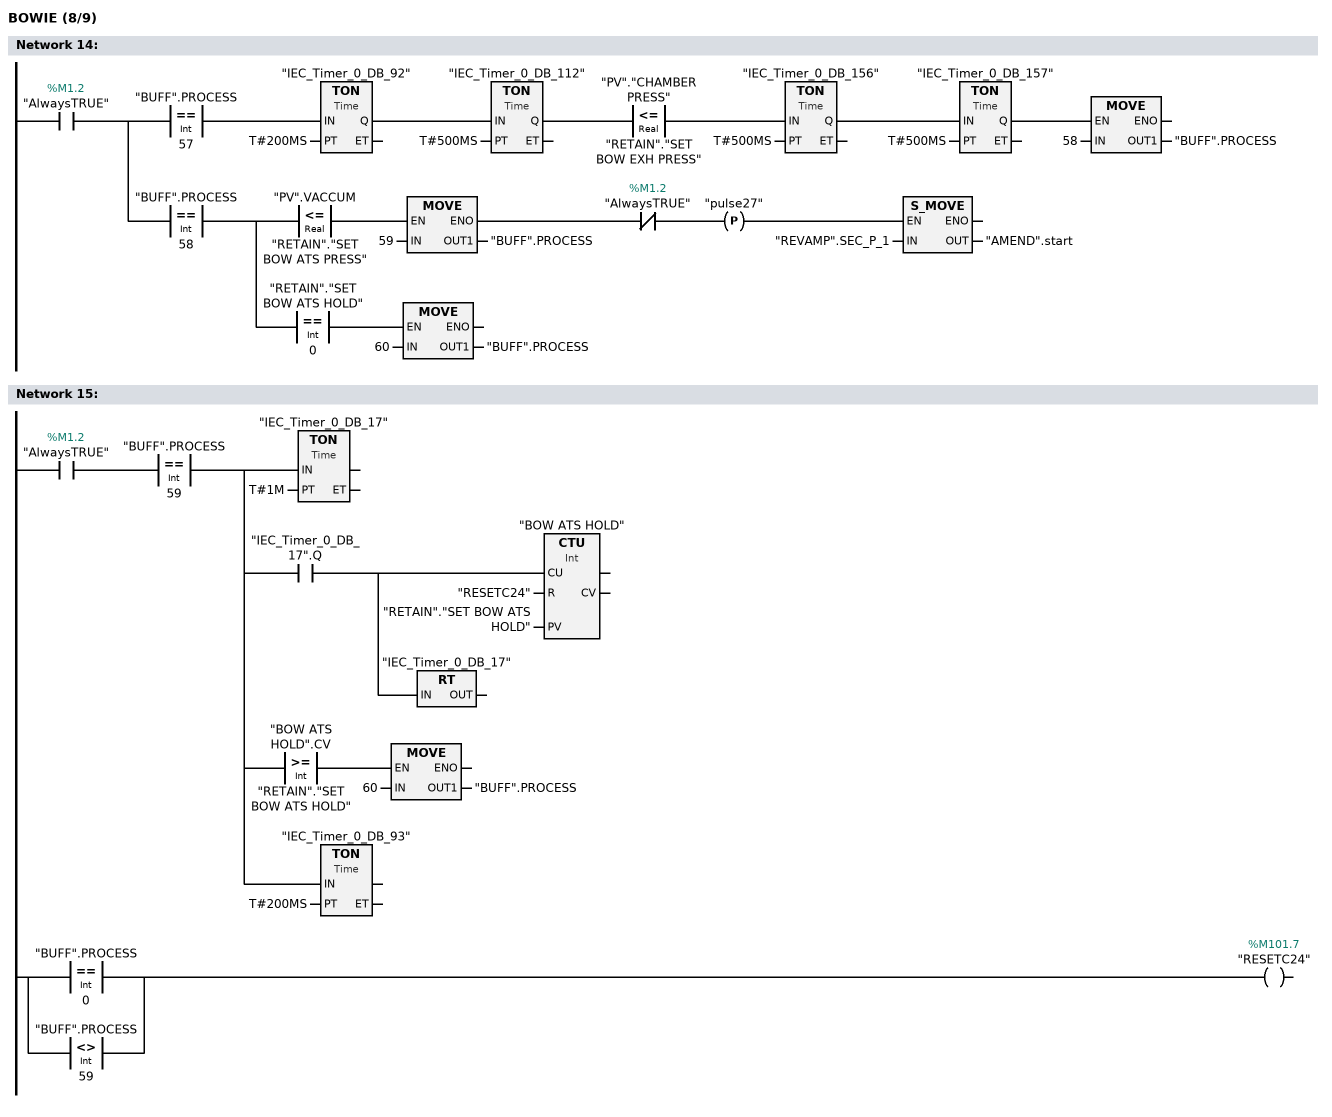
   RUNG wire#powerrail
      Contact( "AlwaysTRUE" )
      wire#w1
      { S7_Templates := "SrcType := Int" } EQ_Contact(in1 := "BUFF".PROCESS, in2 := 57)
      { S7_Templates := "time_type := Time" } "IEC_Timer_0_DB_92".TON(pt := T#200MS, et =>)
      { S7_Templates := "time_type := Time" } "IEC_Timer_0_DB_112".TON(pt := T#500MS, et =>)
      { S7_Templates := "SrcType := Real" } LE_Contact(in1 := "PV"."CHAMBER PRESS", in2 := "RETAIN"."SET BOW EXH PRESS")
      { S7_Templates := "time_type := Time" } "IEC_Timer_0_DB_156".TON(pt := T#500MS, et =>)
      { S7_Templates := "time_type := Time" } "IEC_Timer_0_DB_157".TON(pt := T#500MS, et =>)
      Move(in := 58, out1 => "BUFF".PROCESS)
   END_RUNG
   RUNG wire#w1
      { S7_Templates := "SrcType := Int" } EQ_Contact(in1 := "BUFF".PROCESS, in2 := 58)
      wire#w2
      { S7_Templates := "SrcType := Real" } LE_Contact(in1 := "PV".VACCUM, in2 := "RETAIN"."SET BOW ATS PRESS")
      Move(in := 59, out1 => "BUFF".PROCESS)
      I_Contact( "AlwaysTRUE" )
      P_Trig( "pulse27" )
      S_Move(in := "REVAMP".SEC_P_1, out => "AMEND".start)
   END_RUNG
   RUNG wire#w2
      { S7_Templates := "SrcType := Int" } EQ_Contact(in1 := "RETAIN"."SET BOW ATS HOLD", in2 := 0)
      Move(in := 60, out1 => "BUFF".PROCESS)
   END_RUNG
   // the same network as SCL:
   "IEC_Timer_0_DB_92".TON(IN := "AlwaysTRUE" AND ("BUFF".PROCESS = 57), PT := T#200MS);
   "IEC_Timer_0_DB_112".TON(IN := "IEC_Timer_0_DB_92".Q, PT := T#500MS);
   "IEC_Timer_0_DB_156".TON(IN := "IEC_Timer_0_DB_112".Q AND ("PV"."CHAMBER PRESS" <= "RETAIN"."SET BOW EXH PRESS"),
                           PT := T#500MS);
   "IEC_Timer_0_DB_157".TON(IN := "IEC_Timer_0_DB_156".Q, PT := T#500MS);
   IF "IEC_Timer_0_DB_157".Q THEN "BUFF".PROCESS := 58; END_IF;
   #_w1 := "AlwaysTRUE" AND ("BUFF".PROCESS = 58);
   #_w2 := #_w1 AND ("PV".VACCUM <= "RETAIN"."SET BOW ATS PRESS");
   IF #_w2 THEN "BUFF".PROCESS := 59; END_IF;
   #_w3 := #_w2 AND NOT "AlwaysTRUE";
   #_w4 := #_w3 AND NOT "pulse27";   // rising edge
   "pulse27" := #_w3;
   IF #_w4 THEN "AMEND".start := "REVAMP".SEC_P_1; END_IF;
   IF #_w1 AND ("RETAIN"."SET BOW ATS HOLD" = 0) THEN "BUFF".PROCESS := 60; END_IF;
END_REGION

REGION Network 15
   RUNG wire#powerrail
      Contact( "AlwaysTRUE" )
      { S7_Templates := "SrcType := Int" } EQ_Contact(in1 := "BUFF".PROCESS, in2 := 59)
      wire#w1
      { S7_Templates := "time_type := Time" } "IEC_Timer_0_DB_17".TON(pt := T#1M, et =>)
   END_RUNG
   RUNG wire#w1
      Contact( "IEC_Timer_0_DB_17".Q )
      wire#w2
      { S7_Templates := "value_type := Int" } "BOW ATS HOLD".CTU(r := "RESETC24", pv := "RETAIN"."SET BOW ATS HOLD", cv =>)
   END_RUNG
   RUNG wire#w2
      RT_Coil( "IEC_Timer_0_DB_17" )
   END_RUNG
   RUNG wire#w1
      { S7_Templates := "SrcType := Int" } GE_Contact(in1 := "BOW ATS HOLD".CV, in2 := "RETAIN"."SET BOW ATS HOLD")
      Move(in := 60, out1 => "BUFF".PROCESS)
   END_RUNG
   RUNG wire#w1
      { S7_Templates := "time_type := Time" } "IEC_Timer_0_DB_93".TON(pt := T#200MS, et =>)
   END_RUNG
   RUNG wire#powerrail
      { S7_Templates := "SrcType := Int" } EQ_Contact(in1 := "BUFF".PROCESS, in2 := 0)
      wire#w3
      Coil( "RESETC24" )
   END_RUNG
   RUNG wire#powerrail
      { S7_Templates := "SrcType := Int" } NE_Contact(in1 := "BUFF".PROCESS, in2 := 59)
   END_RUNG wire#w3
   // the same network as SCL:
   #_w1 := "AlwaysTRUE" AND ("BUFF".PROCESS = 59);
   "IEC_Timer_0_DB_17".TON(IN := #_w1, PT := T#1M);
   #_w2 := #_w1 AND "IEC_Timer_0_DB_17".Q;
   "BOW ATS HOLD".CTU(CU := #_w2, R := "RESETC24", PV := "RETAIN"."SET BOW ATS HOLD");
   IF #_w2 THEN RESET_TIMER("IEC_Timer_0_DB_17"); END_IF;
   IF #_w1 AND ("BOW ATS HOLD".CV >= "RETAIN"."SET BOW ATS HOLD") THEN "BUFF".PROCESS := 60; END_IF;
   "IEC_Timer_0_DB_93".TON(IN := #_w1, PT := T#200MS);
   "RESETC24" := ("BUFF".PROCESS = 0) OR ("BUFF".PROCESS <> 59);
END_REGION

REGION Network 16
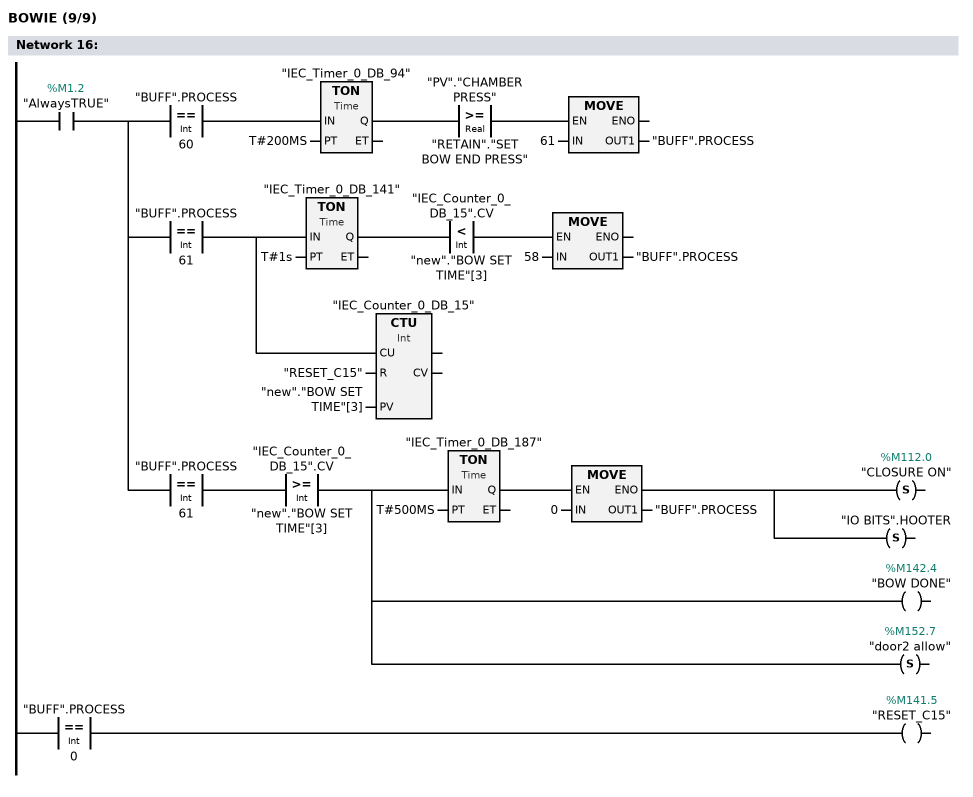
   RUNG wire#powerrail
      Contact( "AlwaysTRUE" )
      wire#w1
      { S7_Templates := "SrcType := Int" } EQ_Contact(in1 := "BUFF".PROCESS, in2 := 60)
      { S7_Templates := "time_type := Time" } "IEC_Timer_0_DB_94".TON(pt := T#200MS, et =>)
      { S7_Templates := "SrcType := Real" } GE_Contact(in1 := "PV"."CHAMBER PRESS", in2 := "RETAIN"."SET BOW END PRESS")
      Move(in := 61, out1 => "BUFF".PROCESS)
   END_RUNG
   RUNG wire#w1
      { S7_Templates := "SrcType := Int" } EQ_Contact(in1 := "BUFF".PROCESS, in2 := 61)
      wire#w2
      { S7_Templates := "time_type := Time" } "IEC_Timer_0_DB_141".TON(pt := T#1s, et =>)
      { S7_Templates := "SrcType := Int" } LT_Contact(in1 := "IEC_Counter_0_DB_15".CV, in2 := "new"."BOW SET TIME"[3])
      Move(in := 58, out1 => "BUFF".PROCESS)
   END_RUNG
   RUNG wire#w2
      { S7_Templates := "value_type := Int" } "IEC_Counter_0_DB_15".CTU(r := "RESET_C15", pv := "new"."BOW SET TIME"[3], cv =>)
   END_RUNG
   RUNG wire#w1
      { S7_Templates := "SrcType := Int" } EQ_Contact(in1 := "BUFF".PROCESS, in2 := 61)
      { S7_Templates := "SrcType := Int" } GE_Contact(in1 := "IEC_Counter_0_DB_15".CV, in2 := "new"."BOW SET TIME"[3])
      wire#w3
      { S7_Templates := "time_type := Time" } "IEC_Timer_0_DB_187".TON(pt := T#500MS, et =>)
      Move(in := 0, out1 => "BUFF".PROCESS)
      wire#w4
      S_Coil( "CLOSURE ON" )
   END_RUNG
   RUNG wire#w4
      S_Coil( "IO BITS".HOOTER )
   END_RUNG
   RUNG wire#w3
      Coil( "BOW DONE" )
   END_RUNG
   RUNG wire#w3
      S_Coil( "door2 allow" )
   END_RUNG
   RUNG wire#powerrail
      { S7_Templates := "SrcType := Int" } EQ_Contact(in1 := "BUFF".PROCESS, in2 := 0)
      Coil( "RESET_C15" )
   END_RUNG
   // the same network as SCL:
   "IEC_Timer_0_DB_94".TON(IN := "AlwaysTRUE" AND ("BUFF".PROCESS = 60), PT := T#200MS);
   IF "IEC_Timer_0_DB_94".Q AND ("PV"."CHAMBER PRESS" >= "RETAIN"."SET BOW END PRESS") THEN
       "BUFF".PROCESS := 61;
   END_IF;
   #_w1 := "AlwaysTRUE" AND ("BUFF".PROCESS = 61);
   "IEC_Timer_0_DB_141".TON(IN := #_w1, PT := T#1s);
   IF "IEC_Timer_0_DB_141".Q AND ("IEC_Counter_0_DB_15".CV < "new"."BOW SET TIME"[3]) THEN
       "BUFF".PROCESS := 58;
   END_IF;
   "IEC_Counter_0_DB_15".CTU(CU := #_w1, R := "RESET_C15", PV := "new"."BOW SET TIME"[3]);
   #_w2 := "AlwaysTRUE" AND ("BUFF".PROCESS = 61) AND ("IEC_Counter_0_DB_15".CV >= "new"."BOW SET TIME"[3]);
   "IEC_Timer_0_DB_187".TON(IN := #_w2, PT := T#500MS);
   IF "IEC_Timer_0_DB_187".Q THEN
       "BUFF".PROCESS := 0;
       "CLOSURE ON" := TRUE;
       "IO BITS".HOOTER := TRUE;
   END_IF;
   "BOW DONE" := #_w2;
   IF #_w2 THEN "door2 allow" := TRUE; END_IF;
   "RESET_C15" := "BUFF".PROCESS = 0;
END_REGION
END_FUNCTION

FUNCTION "SUBOUT" : Void   // FC16, LAD
{ S7_Optimized_Access := 'TRUE' }
// stored: SetENOAutomatically false
   VAR_TEMP   // added for the SCL form of the ladder/FBD networks
      _w1 : Bool;
      _w2 : Bool;
   END_VAR
BEGIN

REGION Network 1
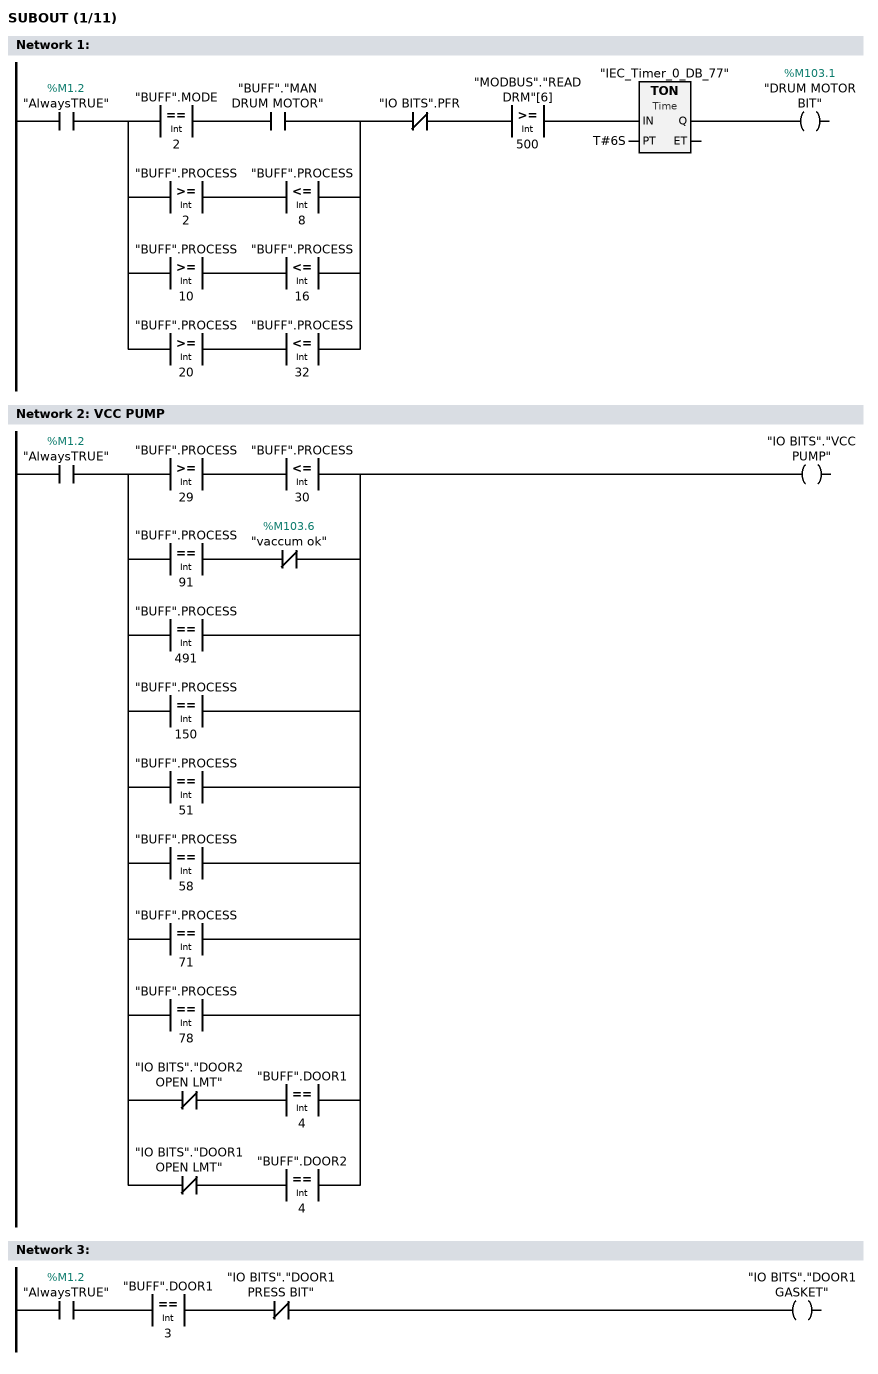
   RUNG wire#powerrail
      Contact( "AlwaysTRUE" )
      wire#w1
      { S7_Templates := "SrcType := Int" } EQ_Contact(in1 := "BUFF".MODE, in2 := 2)
      Contact( "BUFF"."MAN DRUM MOTOR" )
      wire#w2
      I_Contact( "IO BITS".PFR )
      { S7_Templates := "SrcType := Int" } GE_Contact(in1 := "MODBUS"."READ DRM"[6], in2 := 500)
      { S7_Templates := "time_type := Time" } "IEC_Timer_0_DB_77".TON(pt := T#6S, et =>)
      Coil( "DRUM MOTOR BIT" )
   END_RUNG
   RUNG wire#w1
      { S7_Templates := "SrcType := Int" } GE_Contact(in1 := "BUFF".PROCESS, in2 := 2)
      { S7_Templates := "SrcType := Int" } LE_Contact(in1 := "BUFF".PROCESS, in2 := 8)
   END_RUNG wire#w2
   RUNG wire#w1
      { S7_Templates := "SrcType := Int" } GE_Contact(in1 := "BUFF".PROCESS, in2 := 10)
      { S7_Templates := "SrcType := Int" } LE_Contact(in1 := "BUFF".PROCESS, in2 := 16)
   END_RUNG wire#w2
   RUNG wire#w1
      { S7_Templates := "SrcType := Int" } GE_Contact(in1 := "BUFF".PROCESS, in2 := 20)
      { S7_Templates := "SrcType := Int" } LE_Contact(in1 := "BUFF".PROCESS, in2 := 32)
   END_RUNG wire#w2
   // the same network as SCL:
   "IEC_Timer_0_DB_77".TON(IN := "AlwaysTRUE" AND ((("BUFF".MODE = 2) AND "BUFF"."MAN DRUM MOTOR") OR (("BUFF".PROCESS >= 2) AND ("BUFF".PROCESS <= 8)) OR (("BUFF".PROCESS >= 10) AND ("BUFF".PROCESS <= 16)) OR (("BUFF".PROCESS >= 20) AND ("BUFF".PROCESS <= 32))) AND NOT "IO BITS".PFR AND ("MODBUS"."READ DRM"[6] >= 500),
                           PT := T#6S);
   "DRUM MOTOR BIT" := "IEC_Timer_0_DB_77".Q;
END_REGION

REGION Network 2: VCC PUMP
   RUNG wire#powerrail
      Contact( "AlwaysTRUE" )
      wire#w1
      { S7_Templates := "SrcType := Int" } GE_Contact(in1 := "BUFF".PROCESS, in2 := 29)
      { S7_Templates := "SrcType := Int" } LE_Contact(in1 := "BUFF".PROCESS, in2 := 30)
      wire#w2
      Coil( "IO BITS"."VCC PUMP" )
   END_RUNG
   RUNG wire#w1
      { S7_Templates := "SrcType := Int" } EQ_Contact(in1 := "BUFF".PROCESS, in2 := 91)
      I_Contact( "vaccum ok" )
   END_RUNG wire#w2
   RUNG wire#w1
      { S7_Templates := "SrcType := Int" } EQ_Contact(in1 := "BUFF".PROCESS, in2 := 491)
   END_RUNG wire#w2
   RUNG wire#w1
      { S7_Templates := "SrcType := Int" } EQ_Contact(in1 := "BUFF".PROCESS, in2 := 150)
   END_RUNG wire#w2
   RUNG wire#w1
      { S7_Templates := "SrcType := Int" } EQ_Contact(in1 := "BUFF".PROCESS, in2 := 51)
   END_RUNG wire#w2
   RUNG wire#w1
      { S7_Templates := "SrcType := Int" } EQ_Contact(in1 := "BUFF".PROCESS, in2 := 58)
   END_RUNG wire#w2
   RUNG wire#w1
      { S7_Templates := "SrcType := Int" } EQ_Contact(in1 := "BUFF".PROCESS, in2 := 71)
   END_RUNG wire#w2
   RUNG wire#w1
      { S7_Templates := "SrcType := Int" } EQ_Contact(in1 := "BUFF".PROCESS, in2 := 78)
   END_RUNG wire#w2
   RUNG wire#w1
      I_Contact( "IO BITS"."DOOR2 OPEN LMT" )
      { S7_Templates := "SrcType := Int" } EQ_Contact(in1 := "BUFF".DOOR1, in2 := 4)
   END_RUNG wire#w2
   RUNG wire#w1
      I_Contact( "IO BITS"."DOOR1 OPEN LMT" )
      { S7_Templates := "SrcType := Int" } EQ_Contact(in1 := "BUFF".DOOR2, in2 := 4)
   END_RUNG wire#w2
   // the same network as SCL:
   "IO BITS"."VCC PUMP" := "AlwaysTRUE" AND ((("BUFF".PROCESS >= 29) AND ("BUFF".PROCESS <= 30)) OR (("BUFF".PROCESS = 91) AND NOT "vaccum ok") OR ("BUFF".PROCESS = 491) OR ("BUFF".PROCESS = 150) OR ("BUFF".PROCESS = 51) OR ("BUFF".PROCESS = 58) OR ("BUFF".PROCESS = 71) OR ("BUFF".PROCESS = 78) OR (NOT "IO BITS"."DOOR2 OPEN LMT" AND ("BUFF".DOOR1 = 4)) OR (NOT "IO BITS"."DOOR1 OPEN LMT" AND ("BUFF".DOOR2 = 4)));
END_REGION

REGION Network 3
   RUNG wire#powerrail
      Contact( "AlwaysTRUE" )
      { S7_Templates := "SrcType := Int" } EQ_Contact(in1 := "BUFF".DOOR1, in2 := 3)
      I_Contact( "IO BITS"."DOOR1 PRESS BIT" )
      Coil( "IO BITS"."DOOR1 GASKET" )
   END_RUNG
   // the same network as SCL:
   "IO BITS"."DOOR1 GASKET" := "AlwaysTRUE" AND ("BUFF".DOOR1 = 3) AND NOT "IO BITS"."DOOR1 PRESS BIT";
END_REGION

REGION Network 4
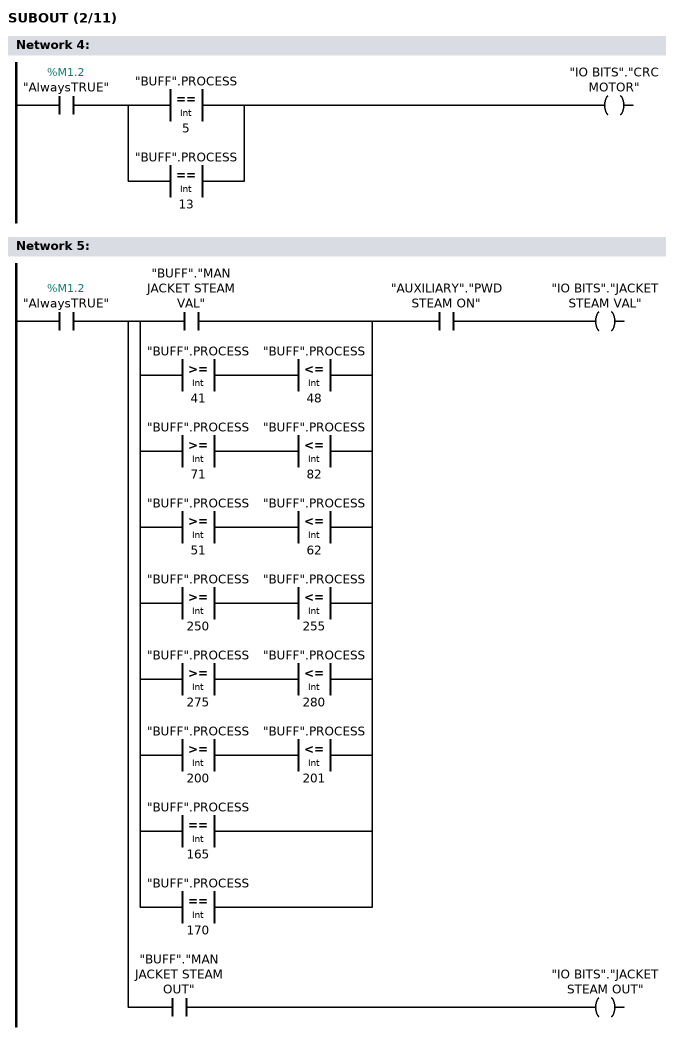
   RUNG wire#powerrail
      Contact( "AlwaysTRUE" )
      wire#w1
      { S7_Templates := "SrcType := Int" } EQ_Contact(in1 := "BUFF".PROCESS, in2 := 5)
      wire#w2
      Coil( "IO BITS"."CRC MOTOR" )
   END_RUNG
   RUNG wire#w1
      { S7_Templates := "SrcType := Int" } EQ_Contact(in1 := "BUFF".PROCESS, in2 := 13)
   END_RUNG wire#w2
   // the same network as SCL:
   "IO BITS"."CRC MOTOR" := "AlwaysTRUE" AND (("BUFF".PROCESS = 5) OR ("BUFF".PROCESS = 13));
END_REGION

REGION Network 5
   RUNG wire#powerrail
      Contact( "AlwaysTRUE" )
      wire#w1
      Contact( "BUFF"."MAN JACKET STEAM VAL" )
      wire#w2
      Contact( "AUXILIARY"."PWD STEAM ON" )
      Coil( "IO BITS"."JACKET STEAM VAL" )
   END_RUNG
   RUNG wire#w1
      { S7_Templates := "SrcType := Int" } GE_Contact(in1 := "BUFF".PROCESS, in2 := 41)
      { S7_Templates := "SrcType := Int" } LE_Contact(in1 := "BUFF".PROCESS, in2 := 48)
   END_RUNG wire#w2
   RUNG wire#w1
      { S7_Templates := "SrcType := Int" } GE_Contact(in1 := "BUFF".PROCESS, in2 := 71)
      { S7_Templates := "SrcType := Int" } LE_Contact(in1 := "BUFF".PROCESS, in2 := 82)
   END_RUNG wire#w2
   RUNG wire#w1
      { S7_Templates := "SrcType := Int" } GE_Contact(in1 := "BUFF".PROCESS, in2 := 51)
      { S7_Templates := "SrcType := Int" } LE_Contact(in1 := "BUFF".PROCESS, in2 := 62)
   END_RUNG wire#w2
   RUNG wire#w1
      { S7_Templates := "SrcType := Int" } GE_Contact(in1 := "BUFF".PROCESS, in2 := 250)
      { S7_Templates := "SrcType := Int" } LE_Contact(in1 := "BUFF".PROCESS, in2 := 255)
   END_RUNG wire#w2
   RUNG wire#w1
      { S7_Templates := "SrcType := Int" } GE_Contact(in1 := "BUFF".PROCESS, in2 := 275)
      { S7_Templates := "SrcType := Int" } LE_Contact(in1 := "BUFF".PROCESS, in2 := 280)
   END_RUNG wire#w2
   RUNG wire#w1
      { S7_Templates := "SrcType := Int" } GE_Contact(in1 := "BUFF".PROCESS, in2 := 200)
      { S7_Templates := "SrcType := Int" } LE_Contact(in1 := "BUFF".PROCESS, in2 := 201)
   END_RUNG wire#w2
   RUNG wire#w1
      { S7_Templates := "SrcType := Int" } EQ_Contact(in1 := "BUFF".PROCESS, in2 := 165)
   END_RUNG wire#w2
   RUNG wire#w1
      { S7_Templates := "SrcType := Int" } EQ_Contact(in1 := "BUFF".PROCESS, in2 := 170)
   END_RUNG wire#w2
   RUNG wire#w1
      Contact( "BUFF"."MAN JACKET STEAM OUT" )
      Coil( "IO BITS"."JACKET STEAM OUT" )
   END_RUNG
   // the same network as SCL:
   "IO BITS"."JACKET STEAM VAL" := "AlwaysTRUE" AND ("BUFF"."MAN JACKET STEAM VAL" OR (("BUFF".PROCESS >= 41) AND ("BUFF".PROCESS <= 48)) OR (("BUFF".PROCESS >= 71) AND ("BUFF".PROCESS <= 82)) OR (("BUFF".PROCESS >= 51) AND ("BUFF".PROCESS <= 62)) OR (("BUFF".PROCESS >= 250) AND ("BUFF".PROCESS <= 255)) OR (("BUFF".PROCESS >= 275) AND ("BUFF".PROCESS <= 280)) OR (("BUFF".PROCESS >= 200) AND ("BUFF".PROCESS <= 201)) OR ("BUFF".PROCESS = 165) OR ("BUFF".PROCESS = 170)) AND "AUXILIARY"."PWD STEAM ON";
   "IO BITS"."JACKET STEAM OUT" := "AlwaysTRUE" AND "BUFF"."MAN JACKET STEAM OUT";
END_REGION

REGION Network 6
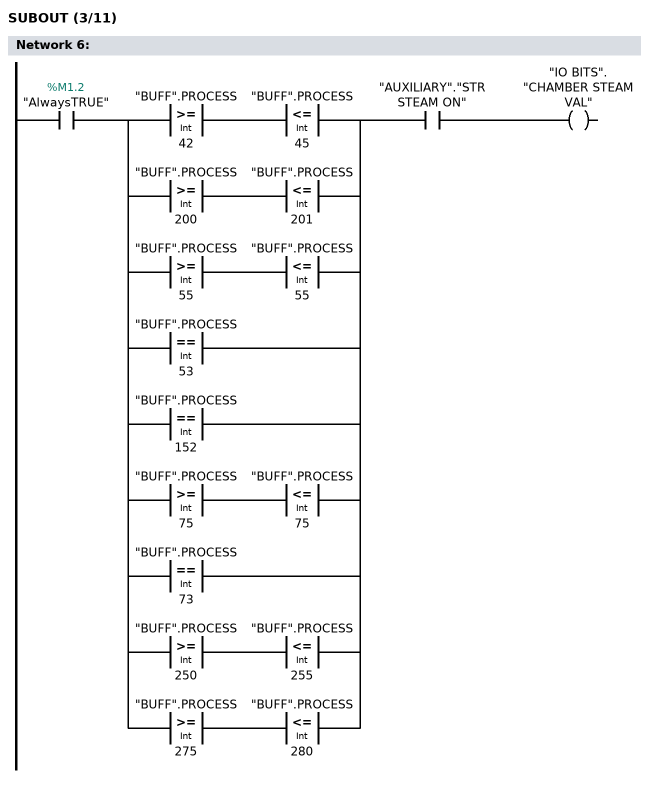
   RUNG wire#powerrail
      Contact( "AlwaysTRUE" )
      wire#w1
      { S7_Templates := "SrcType := Int" } GE_Contact(in1 := "BUFF".PROCESS, in2 := 42)
      { S7_Templates := "SrcType := Int" } LE_Contact(in1 := "BUFF".PROCESS, in2 := 45)
      wire#w2
      Contact( "AUXILIARY"."STR STEAM ON" )
      Coil( "IO BITS"."CHAMBER STEAM VAL" )
   END_RUNG
   RUNG wire#w1
      { S7_Templates := "SrcType := Int" } GE_Contact(in1 := "BUFF".PROCESS, in2 := 200)
      { S7_Templates := "SrcType := Int" } LE_Contact(in1 := "BUFF".PROCESS, in2 := 201)
   END_RUNG wire#w2
   RUNG wire#w1
      { S7_Templates := "SrcType := Int" } GE_Contact(in1 := "BUFF".PROCESS, in2 := 55)
      { S7_Templates := "SrcType := Int" } LE_Contact(in1 := "BUFF".PROCESS, in2 := 55)
   END_RUNG wire#w2
   RUNG wire#w1
      { S7_Templates := "SrcType := Int" } EQ_Contact(in1 := "BUFF".PROCESS, in2 := 53)
   END_RUNG wire#w2
   RUNG wire#w1
      { S7_Templates := "SrcType := Int" } EQ_Contact(in1 := "BUFF".PROCESS, in2 := 152)
   END_RUNG wire#w2
   RUNG wire#w1
      { S7_Templates := "SrcType := Int" } GE_Contact(in1 := "BUFF".PROCESS, in2 := 75)
      { S7_Templates := "SrcType := Int" } LE_Contact(in1 := "BUFF".PROCESS, in2 := 75)
   END_RUNG wire#w2
   RUNG wire#w1
      { S7_Templates := "SrcType := Int" } EQ_Contact(in1 := "BUFF".PROCESS, in2 := 73)
   END_RUNG wire#w2
   RUNG wire#w1
      { S7_Templates := "SrcType := Int" } GE_Contact(in1 := "BUFF".PROCESS, in2 := 250)
      { S7_Templates := "SrcType := Int" } LE_Contact(in1 := "BUFF".PROCESS, in2 := 255)
   END_RUNG wire#w2
   RUNG wire#w1
      { S7_Templates := "SrcType := Int" } GE_Contact(in1 := "BUFF".PROCESS, in2 := 275)
      { S7_Templates := "SrcType := Int" } LE_Contact(in1 := "BUFF".PROCESS, in2 := 280)
   END_RUNG wire#w2
   // the same network as SCL:
   "IO BITS"."CHAMBER STEAM VAL" := "AlwaysTRUE" AND ((("BUFF".PROCESS >= 42) AND ("BUFF".PROCESS <= 45)) OR (("BUFF".PROCESS >= 200) AND ("BUFF".PROCESS <= 201)) OR (("BUFF".PROCESS >= 55) AND ("BUFF".PROCESS <= 55)) OR ("BUFF".PROCESS = 53) OR ("BUFF".PROCESS = 152) OR (("BUFF".PROCESS >= 75) AND ("BUFF".PROCESS <= 75)) OR ("BUFF".PROCESS = 73) OR (("BUFF".PROCESS >= 250) AND ("BUFF".PROCESS <= 255)) OR (("BUFF".PROCESS >= 275) AND ("BUFF".PROCESS <= 280))) AND "AUXILIARY"."STR STEAM ON";
END_REGION

REGION Network 7: CHAMBER EXHAUST VAL
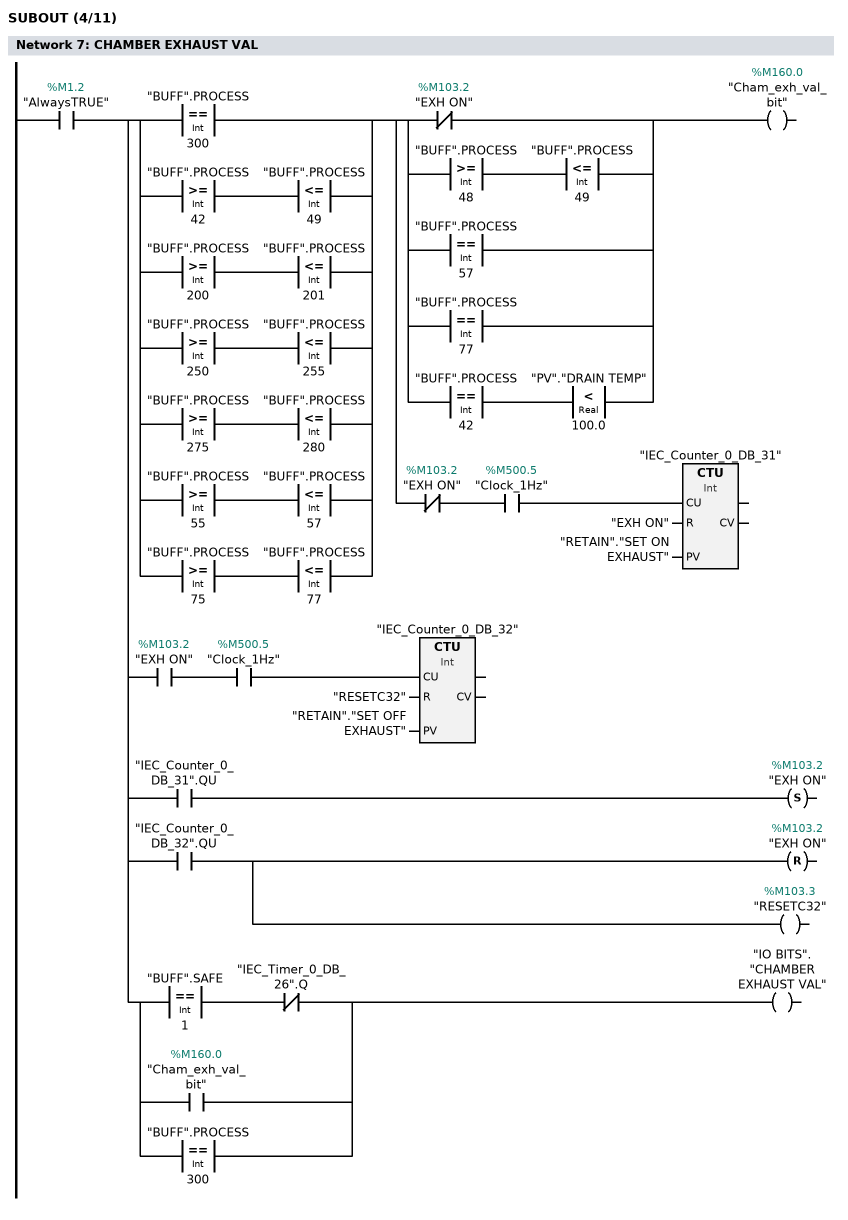
   RUNG wire#powerrail
      Contact( "AlwaysTRUE" )
      wire#w1
      { S7_Templates := "SrcType := Int" } EQ_Contact(in1 := "BUFF".PROCESS, in2 := 300)
      wire#w2
      I_Contact( "EXH ON" )
      wire#w3
      Coil( "Cham_exh_val_bit" )
   END_RUNG
   RUNG wire#w1
      { S7_Templates := "SrcType := Int" } GE_Contact(in1 := "BUFF".PROCESS, in2 := 42)
      { S7_Templates := "SrcType := Int" } LE_Contact(in1 := "BUFF".PROCESS, in2 := 49)
   END_RUNG wire#w2
   RUNG wire#w1
      { S7_Templates := "SrcType := Int" } GE_Contact(in1 := "BUFF".PROCESS, in2 := 200)
      { S7_Templates := "SrcType := Int" } LE_Contact(in1 := "BUFF".PROCESS, in2 := 201)
   END_RUNG wire#w2
   RUNG wire#w1
      { S7_Templates := "SrcType := Int" } GE_Contact(in1 := "BUFF".PROCESS, in2 := 250)
      { S7_Templates := "SrcType := Int" } LE_Contact(in1 := "BUFF".PROCESS, in2 := 255)
   END_RUNG wire#w2
   RUNG wire#w1
      { S7_Templates := "SrcType := Int" } GE_Contact(in1 := "BUFF".PROCESS, in2 := 275)
      { S7_Templates := "SrcType := Int" } LE_Contact(in1 := "BUFF".PROCESS, in2 := 280)
   END_RUNG wire#w2
   RUNG wire#w1
      { S7_Templates := "SrcType := Int" } GE_Contact(in1 := "BUFF".PROCESS, in2 := 55)
      { S7_Templates := "SrcType := Int" } LE_Contact(in1 := "BUFF".PROCESS, in2 := 57)
   END_RUNG wire#w2
   RUNG wire#w1
      { S7_Templates := "SrcType := Int" } GE_Contact(in1 := "BUFF".PROCESS, in2 := 75)
      { S7_Templates := "SrcType := Int" } LE_Contact(in1 := "BUFF".PROCESS, in2 := 77)
   END_RUNG wire#w2
   RUNG wire#w2
      { S7_Templates := "SrcType := Int" } GE_Contact(in1 := "BUFF".PROCESS, in2 := 48)
      { S7_Templates := "SrcType := Int" } LE_Contact(in1 := "BUFF".PROCESS, in2 := 49)
   END_RUNG wire#w3
   RUNG wire#w2
      { S7_Templates := "SrcType := Int" } EQ_Contact(in1 := "BUFF".PROCESS, in2 := 57)
   END_RUNG wire#w3
   RUNG wire#w2
      { S7_Templates := "SrcType := Int" } EQ_Contact(in1 := "BUFF".PROCESS, in2 := 77)
   END_RUNG wire#w3
   RUNG wire#w2
      { S7_Templates := "SrcType := Int" } EQ_Contact(in1 := "BUFF".PROCESS, in2 := 42)
      { S7_Templates := "SrcType := Real" } LT_Contact(in1 := "PV"."DRAIN TEMP", in2 := 100.0)
   END_RUNG wire#w3
   RUNG wire#w2
      I_Contact( "EXH ON" )
      Contact( "Clock_1Hz" )
      { S7_Templates := "value_type := Int" } "IEC_Counter_0_DB_31".CTU(r := "EXH ON", pv := "RETAIN"."SET ON EXHAUST", cv =>)
   END_RUNG
   RUNG wire#w1
      Contact( "EXH ON" )
      Contact( "Clock_1Hz" )
      { S7_Templates := "value_type := Int" } "IEC_Counter_0_DB_32".CTU(r := "RESETC32", pv := "RETAIN"."SET OFF EXHAUST", cv =>)
   END_RUNG
   RUNG wire#w1
      Contact( "IEC_Counter_0_DB_31".QU )
      S_Coil( "EXH ON" )
   END_RUNG
   RUNG wire#w1
      Contact( "IEC_Counter_0_DB_32".QU )
      wire#w4
      R_Coil( "EXH ON" )
   END_RUNG
   RUNG wire#w4
      Coil( "RESETC32" )
   END_RUNG
   RUNG wire#w1
      { S7_Templates := "SrcType := Int" } EQ_Contact(in1 := "BUFF".SAFE, in2 := 1)
      I_Contact( "IEC_Timer_0_DB_26".Q )
      wire#w5
      Coil( "IO BITS"."CHAMBER EXHAUST VAL" )
   END_RUNG
   RUNG wire#w1
      Contact( "Cham_exh_val_bit" )
   END_RUNG wire#w5
   RUNG wire#w1
      { S7_Templates := "SrcType := Int" } EQ_Contact(in1 := "BUFF".PROCESS, in2 := 300)
   END_RUNG wire#w5
   // the same network as SCL:
   #_w1 := "AlwaysTRUE" AND (("BUFF".PROCESS = 300) OR (("BUFF".PROCESS >= 42) AND ("BUFF".PROCESS <= 49)) OR (("BUFF".PROCESS >= 200) AND ("BUFF".PROCESS <= 201)) OR (("BUFF".PROCESS >= 250) AND ("BUFF".PROCESS <= 255)) OR (("BUFF".PROCESS >= 275) AND ("BUFF".PROCESS <= 280)) OR (("BUFF".PROCESS >= 55) AND ("BUFF".PROCESS <= 57)) OR (("BUFF".PROCESS >= 75) AND ("BUFF".PROCESS <= 77)));
   "Cham_exh_val_bit" := #_w1 AND (NOT "EXH ON" OR (("BUFF".PROCESS >= 48) AND ("BUFF".PROCESS <= 49)) OR ("BUFF".PROCESS = 57) OR ("BUFF".PROCESS = 77) OR (("BUFF".PROCESS = 42) AND ("PV"."DRAIN TEMP" < 100.0)));
   "IEC_Counter_0_DB_31".CTU(CU := #_w1 AND NOT "EXH ON" AND "Clock_1Hz",
                           R := "EXH ON",
                           PV := "RETAIN"."SET ON EXHAUST");
   "IEC_Counter_0_DB_32".CTU(CU := "AlwaysTRUE" AND "EXH ON" AND "Clock_1Hz",
                           R := "RESETC32",
                           PV := "RETAIN"."SET OFF EXHAUST");
   IF "AlwaysTRUE" AND "IEC_Counter_0_DB_31".QU THEN "EXH ON" := TRUE; END_IF;
   #_w2 := "AlwaysTRUE" AND "IEC_Counter_0_DB_32".QU;
   IF #_w2 THEN "EXH ON" := FALSE; END_IF;
   "RESETC32" := #_w2;
   "IO BITS"."CHAMBER EXHAUST VAL" := "AlwaysTRUE" AND ((("BUFF".SAFE = 1) AND NOT "IEC_Timer_0_DB_26".Q) OR "Cham_exh_val_bit" OR ("BUFF".PROCESS = 300));
END_REGION

REGION Network 8
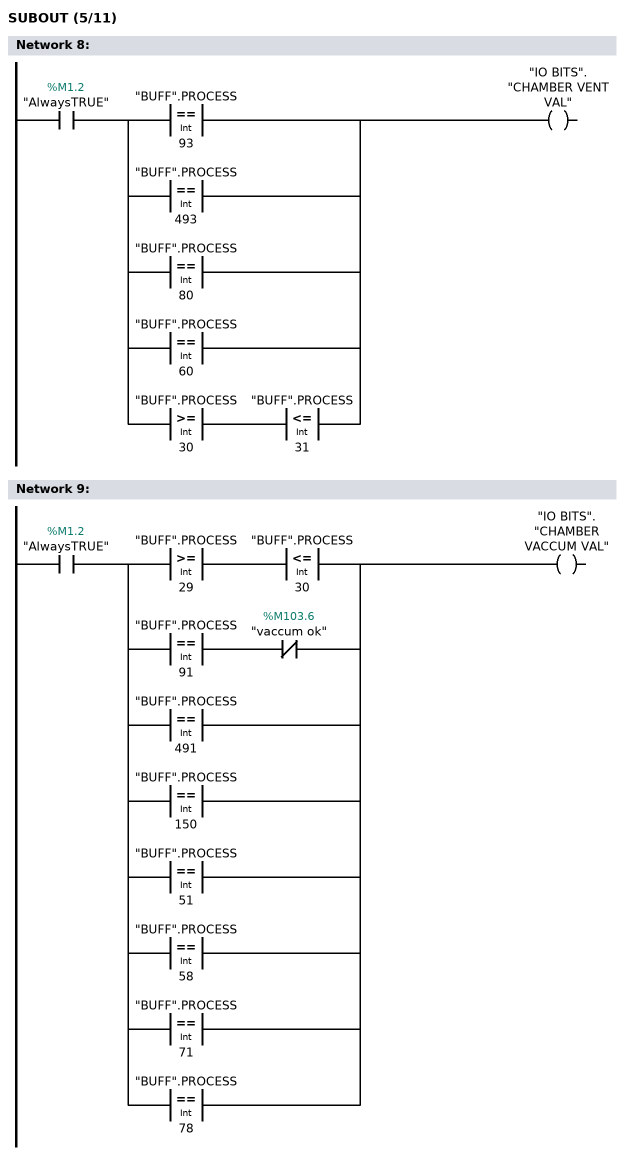
   RUNG wire#powerrail
      Contact( "AlwaysTRUE" )
      wire#w1
      { S7_Templates := "SrcType := Int" } EQ_Contact(in1 := "BUFF".PROCESS, in2 := 93)
      wire#w2
      Coil( "IO BITS"."CHAMBER VENT VAL" )
   END_RUNG
   RUNG wire#w1
      { S7_Templates := "SrcType := Int" } EQ_Contact(in1 := "BUFF".PROCESS, in2 := 493)
   END_RUNG wire#w2
   RUNG wire#w1
      { S7_Templates := "SrcType := Int" } EQ_Contact(in1 := "BUFF".PROCESS, in2 := 80)
   END_RUNG wire#w2
   RUNG wire#w1
      { S7_Templates := "SrcType := Int" } EQ_Contact(in1 := "BUFF".PROCESS, in2 := 60)
   END_RUNG wire#w2
   RUNG wire#w1
      { S7_Templates := "SrcType := Int" } GE_Contact(in1 := "BUFF".PROCESS, in2 := 30)
      { S7_Templates := "SrcType := Int" } LE_Contact(in1 := "BUFF".PROCESS, in2 := 31)
   END_RUNG wire#w2
   // the same network as SCL:
   "IO BITS"."CHAMBER VENT VAL" := "AlwaysTRUE" AND (("BUFF".PROCESS = 93) OR ("BUFF".PROCESS = 493) OR ("BUFF".PROCESS = 80) OR ("BUFF".PROCESS = 60) OR (("BUFF".PROCESS >= 30) AND ("BUFF".PROCESS <= 31)));
END_REGION

REGION Network 9
   RUNG wire#powerrail
      Contact( "AlwaysTRUE" )
      wire#w1
      { S7_Templates := "SrcType := Int" } GE_Contact(in1 := "BUFF".PROCESS, in2 := 29)
      { S7_Templates := "SrcType := Int" } LE_Contact(in1 := "BUFF".PROCESS, in2 := 30)
      wire#w2
      Coil( "IO BITS"."CHAMBER VACCUM VAL" )
   END_RUNG
   RUNG wire#w1
      { S7_Templates := "SrcType := Int" } EQ_Contact(in1 := "BUFF".PROCESS, in2 := 91)
      I_Contact( "vaccum ok" )
   END_RUNG wire#w2
   RUNG wire#w1
      { S7_Templates := "SrcType := Int" } EQ_Contact(in1 := "BUFF".PROCESS, in2 := 491)
   END_RUNG wire#w2
   RUNG wire#w1
      { S7_Templates := "SrcType := Int" } EQ_Contact(in1 := "BUFF".PROCESS, in2 := 150)
   END_RUNG wire#w2
   RUNG wire#w1
      { S7_Templates := "SrcType := Int" } EQ_Contact(in1 := "BUFF".PROCESS, in2 := 51)
   END_RUNG wire#w2
   RUNG wire#w1
      { S7_Templates := "SrcType := Int" } EQ_Contact(in1 := "BUFF".PROCESS, in2 := 58)
   END_RUNG wire#w2
   RUNG wire#w1
      { S7_Templates := "SrcType := Int" } EQ_Contact(in1 := "BUFF".PROCESS, in2 := 71)
   END_RUNG wire#w2
   RUNG wire#w1
      { S7_Templates := "SrcType := Int" } EQ_Contact(in1 := "BUFF".PROCESS, in2 := 78)
   END_RUNG wire#w2
   // the same network as SCL:
   "IO BITS"."CHAMBER VACCUM VAL" := "AlwaysTRUE" AND ((("BUFF".PROCESS >= 29) AND ("BUFF".PROCESS <= 30)) OR (("BUFF".PROCESS = 91) AND NOT "vaccum ok") OR ("BUFF".PROCESS = 491) OR ("BUFF".PROCESS = 150) OR ("BUFF".PROCESS = 51) OR ("BUFF".PROCESS = 58) OR ("BUFF".PROCESS = 71) OR ("BUFF".PROCESS = 78));
END_REGION

REGION Network 10
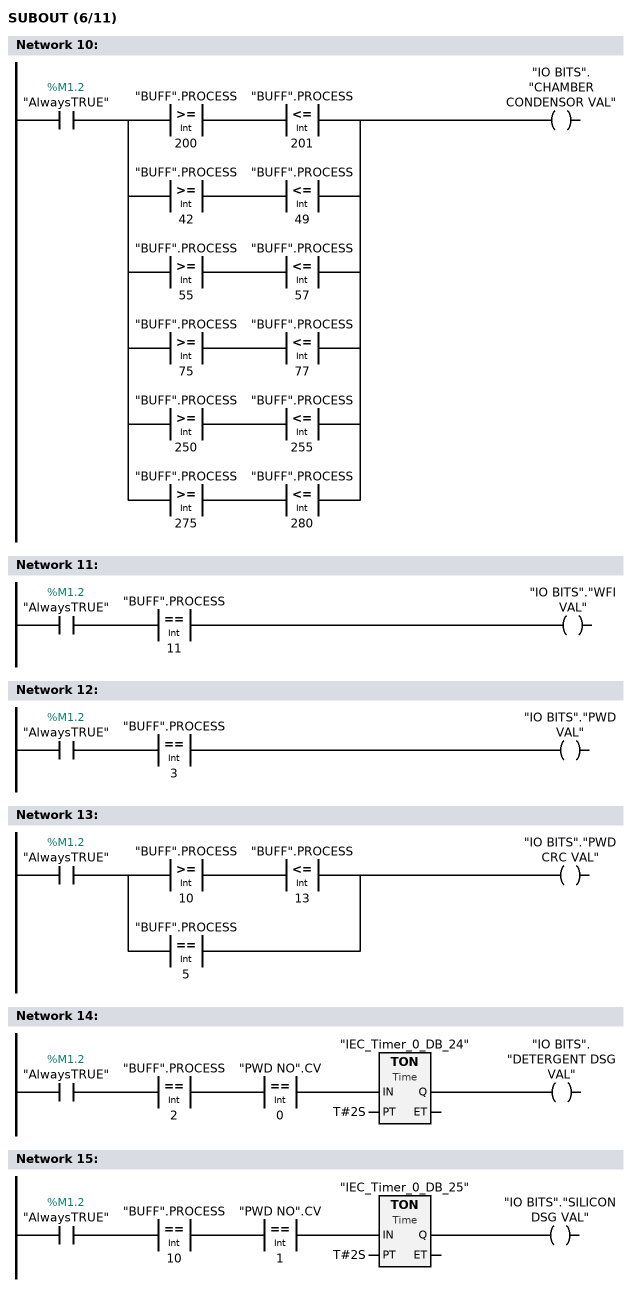
   RUNG wire#powerrail
      Contact( "AlwaysTRUE" )
      wire#w1
      { S7_Templates := "SrcType := Int" } GE_Contact(in1 := "BUFF".PROCESS, in2 := 200)
      { S7_Templates := "SrcType := Int" } LE_Contact(in1 := "BUFF".PROCESS, in2 := 201)
      wire#w2
      Coil( "IO BITS"."CHAMBER CONDENSOR VAL" )
   END_RUNG
   RUNG wire#w1
      { S7_Templates := "SrcType := Int" } GE_Contact(in1 := "BUFF".PROCESS, in2 := 42)
      { S7_Templates := "SrcType := Int" } LE_Contact(in1 := "BUFF".PROCESS, in2 := 49)
   END_RUNG wire#w2
   RUNG wire#w1
      { S7_Templates := "SrcType := Int" } GE_Contact(in1 := "BUFF".PROCESS, in2 := 55)
      { S7_Templates := "SrcType := Int" } LE_Contact(in1 := "BUFF".PROCESS, in2 := 57)
   END_RUNG wire#w2
   RUNG wire#w1
      { S7_Templates := "SrcType := Int" } GE_Contact(in1 := "BUFF".PROCESS, in2 := 75)
      { S7_Templates := "SrcType := Int" } LE_Contact(in1 := "BUFF".PROCESS, in2 := 77)
   END_RUNG wire#w2
   RUNG wire#w1
      { S7_Templates := "SrcType := Int" } GE_Contact(in1 := "BUFF".PROCESS, in2 := 250)
      { S7_Templates := "SrcType := Int" } LE_Contact(in1 := "BUFF".PROCESS, in2 := 255)
   END_RUNG wire#w2
   RUNG wire#w1
      { S7_Templates := "SrcType := Int" } GE_Contact(in1 := "BUFF".PROCESS, in2 := 275)
      { S7_Templates := "SrcType := Int" } LE_Contact(in1 := "BUFF".PROCESS, in2 := 280)
   END_RUNG wire#w2
   // the same network as SCL:
   "IO BITS"."CHAMBER CONDENSOR VAL" := "AlwaysTRUE" AND ((("BUFF".PROCESS >= 200) AND ("BUFF".PROCESS <= 201)) OR (("BUFF".PROCESS >= 42) AND ("BUFF".PROCESS <= 49)) OR (("BUFF".PROCESS >= 55) AND ("BUFF".PROCESS <= 57)) OR (("BUFF".PROCESS >= 75) AND ("BUFF".PROCESS <= 77)) OR (("BUFF".PROCESS >= 250) AND ("BUFF".PROCESS <= 255)) OR (("BUFF".PROCESS >= 275) AND ("BUFF".PROCESS <= 280)));
END_REGION

REGION Network 11
   RUNG wire#powerrail
      Contact( "AlwaysTRUE" )
      { S7_Templates := "SrcType := Int" } EQ_Contact(in1 := "BUFF".PROCESS, in2 := 11)
      Coil( "IO BITS"."WFI VAL" )
   END_RUNG
   // the same network as SCL:
   "IO BITS"."WFI VAL" := "AlwaysTRUE" AND ("BUFF".PROCESS = 11);
END_REGION

REGION Network 12
   RUNG wire#powerrail
      Contact( "AlwaysTRUE" )
      { S7_Templates := "SrcType := Int" } EQ_Contact(in1 := "BUFF".PROCESS, in2 := 3)
      Coil( "IO BITS"."PWD VAL" )
   END_RUNG
   // the same network as SCL:
   "IO BITS"."PWD VAL" := "AlwaysTRUE" AND ("BUFF".PROCESS = 3);
END_REGION

REGION Network 13
   RUNG wire#powerrail
      Contact( "AlwaysTRUE" )
      wire#w1
      { S7_Templates := "SrcType := Int" } GE_Contact(in1 := "BUFF".PROCESS, in2 := 10)
      { S7_Templates := "SrcType := Int" } LE_Contact(in1 := "BUFF".PROCESS, in2 := 13)
      wire#w2
      Coil( "IO BITS"."PWD CRC VAL" )
   END_RUNG
   RUNG wire#w1
      { S7_Templates := "SrcType := Int" } EQ_Contact(in1 := "BUFF".PROCESS, in2 := 5)
   END_RUNG wire#w2
   // the same network as SCL:
   "IO BITS"."PWD CRC VAL" := "AlwaysTRUE" AND ((("BUFF".PROCESS >= 10) AND ("BUFF".PROCESS <= 13)) OR ("BUFF".PROCESS = 5));
END_REGION

REGION Network 14
   RUNG wire#powerrail
      Contact( "AlwaysTRUE" )
      { S7_Templates := "SrcType := Int" } EQ_Contact(in1 := "BUFF".PROCESS, in2 := 2)
      { S7_Templates := "SrcType := Int" } EQ_Contact(in1 := "PWD NO".CV, in2 := 0)
      { S7_Templates := "time_type := Time" } "IEC_Timer_0_DB_24".TON(pt := T#2S, et =>)
      Coil( "IO BITS"."DETERGENT DSG VAL" )
   END_RUNG
   // the same network as SCL:
   "IEC_Timer_0_DB_24".TON(IN := "AlwaysTRUE" AND ("BUFF".PROCESS = 2) AND ("PWD NO".CV = 0), PT := T#2S);
   "IO BITS"."DETERGENT DSG VAL" := "IEC_Timer_0_DB_24".Q;
END_REGION

REGION Network 15
   RUNG wire#powerrail
      Contact( "AlwaysTRUE" )
      { S7_Templates := "SrcType := Int" } EQ_Contact(in1 := "BUFF".PROCESS, in2 := 10)
      { S7_Templates := "SrcType := Int" } EQ_Contact(in1 := "PWD NO".CV, in2 := 1)
      { S7_Templates := "time_type := Time" } "IEC_Timer_0_DB_25".TON(pt := T#2S, et =>)
      Coil( "IO BITS"."SILICON DSG VAL" )
   END_RUNG
   // the same network as SCL:
   "IEC_Timer_0_DB_25".TON(IN := "AlwaysTRUE" AND ("BUFF".PROCESS = 10) AND ("PWD NO".CV = 1), PT := T#2S);
   "IO BITS"."SILICON DSG VAL" := "IEC_Timer_0_DB_25".Q;
END_REGION

REGION Network 16: DRAIN VAL
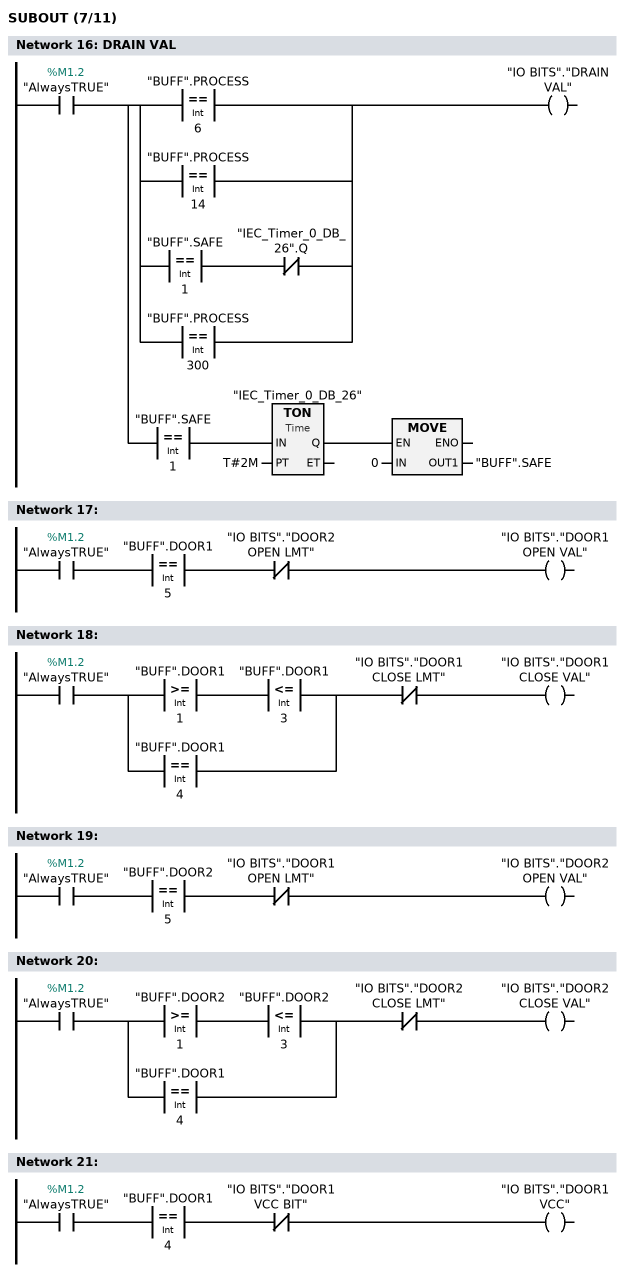
   RUNG wire#powerrail
      Contact( "AlwaysTRUE" )
      wire#w1
      { S7_Templates := "SrcType := Int" } EQ_Contact(in1 := "BUFF".PROCESS, in2 := 6)
      wire#w2
      Coil( "IO BITS"."DRAIN VAL" )
   END_RUNG
   RUNG wire#w1
      { S7_Templates := "SrcType := Int" } EQ_Contact(in1 := "BUFF".PROCESS, in2 := 14)
   END_RUNG wire#w2
   RUNG wire#w1
      { S7_Templates := "SrcType := Int" } EQ_Contact(in1 := "BUFF".SAFE, in2 := 1)
      I_Contact( "IEC_Timer_0_DB_26".Q )
   END_RUNG wire#w2
   RUNG wire#w1
      { S7_Templates := "SrcType := Int" } EQ_Contact(in1 := "BUFF".PROCESS, in2 := 300)
   END_RUNG wire#w2
   RUNG wire#w1
      { S7_Templates := "SrcType := Int" } EQ_Contact(in1 := "BUFF".SAFE, in2 := 1)
      { S7_Templates := "time_type := Time" } "IEC_Timer_0_DB_26".TON(pt := T#2M, et =>)
      Move(in := 0, out1 => "BUFF".SAFE)
   END_RUNG
   // the same network as SCL:
   "IO BITS"."DRAIN VAL" := "AlwaysTRUE" AND (("BUFF".PROCESS = 6) OR ("BUFF".PROCESS = 14) OR (("BUFF".SAFE = 1) AND NOT "IEC_Timer_0_DB_26".Q) OR ("BUFF".PROCESS = 300));
   "IEC_Timer_0_DB_26".TON(IN := "AlwaysTRUE" AND ("BUFF".SAFE = 1), PT := T#2M);
   IF "IEC_Timer_0_DB_26".Q THEN "BUFF".SAFE := 0; END_IF;
END_REGION

REGION Network 17
   RUNG wire#powerrail
      Contact( "AlwaysTRUE" )
      { S7_Templates := "SrcType := Int" } EQ_Contact(in1 := "BUFF".DOOR1, in2 := 5)
      I_Contact( "IO BITS"."DOOR2 OPEN LMT" )
      Coil( "IO BITS"."DOOR1 OPEN VAL" )
   END_RUNG
   // the same network as SCL:
   "IO BITS"."DOOR1 OPEN VAL" := "AlwaysTRUE" AND ("BUFF".DOOR1 = 5) AND NOT "IO BITS"."DOOR2 OPEN LMT";
END_REGION

REGION Network 18
   RUNG wire#powerrail
      Contact( "AlwaysTRUE" )
      wire#w1
      { S7_Templates := "SrcType := Int" } GE_Contact(in1 := "BUFF".DOOR1, in2 := 1)
      { S7_Templates := "SrcType := Int" } LE_Contact(in1 := "BUFF".DOOR1, in2 := 3)
      wire#w2
      I_Contact( "IO BITS"."DOOR1 CLOSE LMT" )
      Coil( "IO BITS"."DOOR1 CLOSE VAL" )
   END_RUNG
   RUNG wire#w1
      { S7_Templates := "SrcType := Int" } EQ_Contact(in1 := "BUFF".DOOR1, in2 := 4)
   END_RUNG wire#w2
   // the same network as SCL:
   "IO BITS"."DOOR1 CLOSE VAL" := "AlwaysTRUE" AND ((("BUFF".DOOR1 >= 1) AND ("BUFF".DOOR1 <= 3)) OR ("BUFF".DOOR1 = 4)) AND NOT "IO BITS"."DOOR1 CLOSE LMT";
END_REGION

REGION Network 19
   RUNG wire#powerrail
      Contact( "AlwaysTRUE" )
      { S7_Templates := "SrcType := Int" } EQ_Contact(in1 := "BUFF".DOOR2, in2 := 5)
      I_Contact( "IO BITS"."DOOR1 OPEN LMT" )
      Coil( "IO BITS"."DOOR2 OPEN VAL" )
   END_RUNG
   // the same network as SCL:
   "IO BITS"."DOOR2 OPEN VAL" := "AlwaysTRUE" AND ("BUFF".DOOR2 = 5) AND NOT "IO BITS"."DOOR1 OPEN LMT";
END_REGION

REGION Network 20
   RUNG wire#powerrail
      Contact( "AlwaysTRUE" )
      wire#w1
      { S7_Templates := "SrcType := Int" } GE_Contact(in1 := "BUFF".DOOR2, in2 := 1)
      { S7_Templates := "SrcType := Int" } LE_Contact(in1 := "BUFF".DOOR2, in2 := 3)
      wire#w2
      I_Contact( "IO BITS"."DOOR2 CLOSE LMT" )
      Coil( "IO BITS"."DOOR2 CLOSE VAL" )
   END_RUNG
   RUNG wire#w1
      { S7_Templates := "SrcType := Int" } EQ_Contact(in1 := "BUFF".DOOR1, in2 := 4)
   END_RUNG wire#w2
   // the same network as SCL:
   "IO BITS"."DOOR2 CLOSE VAL" := "AlwaysTRUE" AND ((("BUFF".DOOR2 >= 1) AND ("BUFF".DOOR2 <= 3)) OR ("BUFF".DOOR1 = 4)) AND NOT "IO BITS"."DOOR2 CLOSE LMT";
END_REGION

REGION Network 21
   RUNG wire#powerrail
      Contact( "AlwaysTRUE" )
      { S7_Templates := "SrcType := Int" } EQ_Contact(in1 := "BUFF".DOOR1, in2 := 4)
      I_Contact( "IO BITS"."DOOR1 VCC BIT" )
      Coil( "IO BITS"."DOOR1 VCC" )
   END_RUNG
   // the same network as SCL:
   "IO BITS"."DOOR1 VCC" := "AlwaysTRUE" AND ("BUFF".DOOR1 = 4) AND NOT "IO BITS"."DOOR1 VCC BIT";
END_REGION

REGION Network 22
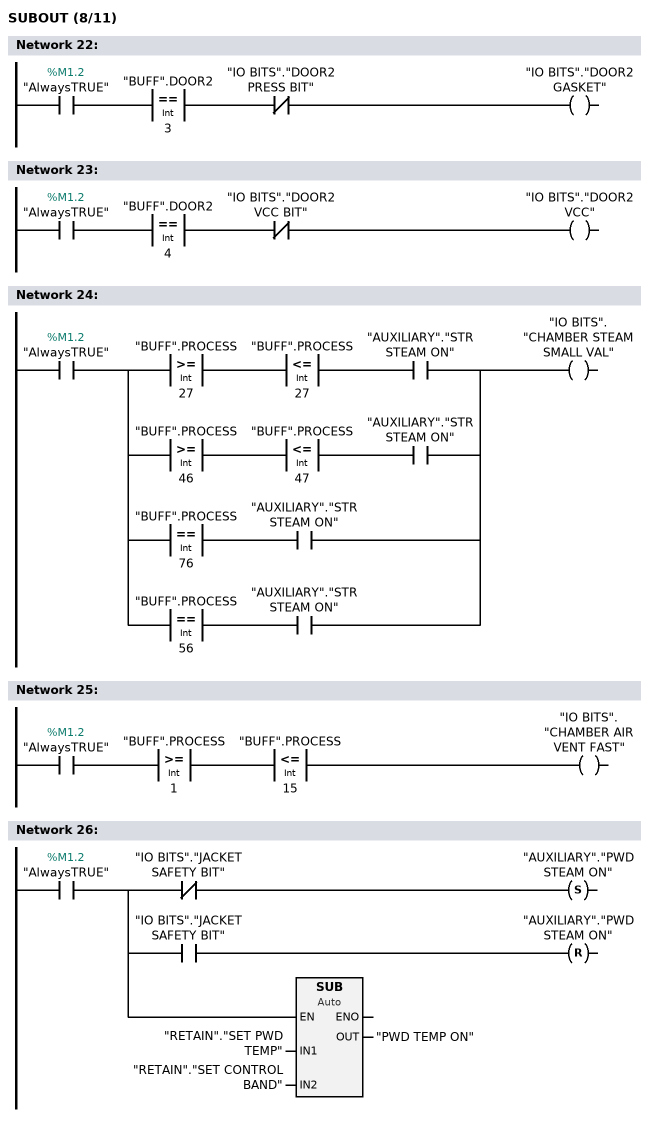
   RUNG wire#powerrail
      Contact( "AlwaysTRUE" )
      { S7_Templates := "SrcType := Int" } EQ_Contact(in1 := "BUFF".DOOR2, in2 := 3)
      I_Contact( "IO BITS"."DOOR2 PRESS BIT" )
      Coil( "IO BITS"."DOOR2 GASKET" )
   END_RUNG
   // the same network as SCL:
   "IO BITS"."DOOR2 GASKET" := "AlwaysTRUE" AND ("BUFF".DOOR2 = 3) AND NOT "IO BITS"."DOOR2 PRESS BIT";
END_REGION

REGION Network 23
   RUNG wire#powerrail
      Contact( "AlwaysTRUE" )
      { S7_Templates := "SrcType := Int" } EQ_Contact(in1 := "BUFF".DOOR2, in2 := 4)
      I_Contact( "IO BITS"."DOOR2 VCC BIT" )
      Coil( "IO BITS"."DOOR2 VCC" )
   END_RUNG
   // the same network as SCL:
   "IO BITS"."DOOR2 VCC" := "AlwaysTRUE" AND ("BUFF".DOOR2 = 4) AND NOT "IO BITS"."DOOR2 VCC BIT";
END_REGION

REGION Network 24
   RUNG wire#powerrail
      Contact( "AlwaysTRUE" )
      wire#w1
      { S7_Templates := "SrcType := Int" } GE_Contact(in1 := "BUFF".PROCESS, in2 := 27)
      { S7_Templates := "SrcType := Int" } LE_Contact(in1 := "BUFF".PROCESS, in2 := 27)
      Contact( "AUXILIARY"."STR STEAM ON" )
      wire#w2
      Coil( "IO BITS"."CHAMBER STEAM SMALL VAL" )
   END_RUNG
   RUNG wire#w1
      { S7_Templates := "SrcType := Int" } GE_Contact(in1 := "BUFF".PROCESS, in2 := 46)
      { S7_Templates := "SrcType := Int" } LE_Contact(in1 := "BUFF".PROCESS, in2 := 47)
      Contact( "AUXILIARY"."STR STEAM ON" )
   END_RUNG wire#w2
   RUNG wire#w1
      { S7_Templates := "SrcType := Int" } EQ_Contact(in1 := "BUFF".PROCESS, in2 := 76)
      Contact( "AUXILIARY"."STR STEAM ON" )
   END_RUNG wire#w2
   RUNG wire#w1
      { S7_Templates := "SrcType := Int" } EQ_Contact(in1 := "BUFF".PROCESS, in2 := 56)
      Contact( "AUXILIARY"."STR STEAM ON" )
   END_RUNG wire#w2
   // the same network as SCL:
   "IO BITS"."CHAMBER STEAM SMALL VAL" := "AlwaysTRUE" AND ((("BUFF".PROCESS >= 27) AND ("BUFF".PROCESS <= 27) AND "AUXILIARY"."STR STEAM ON") OR (("BUFF".PROCESS >= 46) AND ("BUFF".PROCESS <= 47) AND "AUXILIARY"."STR STEAM ON") OR (("BUFF".PROCESS = 76) AND "AUXILIARY"."STR STEAM ON") OR (("BUFF".PROCESS = 56) AND "AUXILIARY"."STR STEAM ON"));
END_REGION

REGION Network 25
   RUNG wire#powerrail
      Contact( "AlwaysTRUE" )
      { S7_Templates := "SrcType := Int" } GE_Contact(in1 := "BUFF".PROCESS, in2 := 1)
      { S7_Templates := "SrcType := Int" } LE_Contact(in1 := "BUFF".PROCESS, in2 := 15)
      Coil( "IO BITS"."CHAMBER AIR VENT FAST" )
   END_RUNG
   // the same network as SCL:
   "IO BITS"."CHAMBER AIR VENT FAST" := "AlwaysTRUE" AND ("BUFF".PROCESS >= 1) AND ("BUFF".PROCESS <= 15);
END_REGION

REGION Network 26
   RUNG wire#powerrail
      Contact( "AlwaysTRUE" )
      wire#w1
      I_Contact( "IO BITS"."JACKET SAFETY BIT" )
      S_Coil( "AUXILIARY"."PWD STEAM ON" )
   END_RUNG
   RUNG wire#w1
      Contact( "IO BITS"."JACKET SAFETY BIT" )
      R_Coil( "AUXILIARY"."PWD STEAM ON" )
   END_RUNG
   RUNG wire#w1
      Sub(in1 := "RETAIN"."SET PWD TEMP", in2 := "RETAIN"."SET CONTROL BAND", out => "PWD TEMP ON")
   END_RUNG
   // the same network as SCL:
   IF "AlwaysTRUE" AND NOT "IO BITS"."JACKET SAFETY BIT" THEN "AUXILIARY"."PWD STEAM ON" := TRUE; END_IF;
   IF "AlwaysTRUE" AND "IO BITS"."JACKET SAFETY BIT" THEN "AUXILIARY"."PWD STEAM ON" := FALSE; END_IF;
   IF "AlwaysTRUE" THEN "PWD TEMP ON" := "RETAIN"."SET PWD TEMP" - "RETAIN"."SET CONTROL BAND"; END_IF;
END_REGION

REGION Network 27
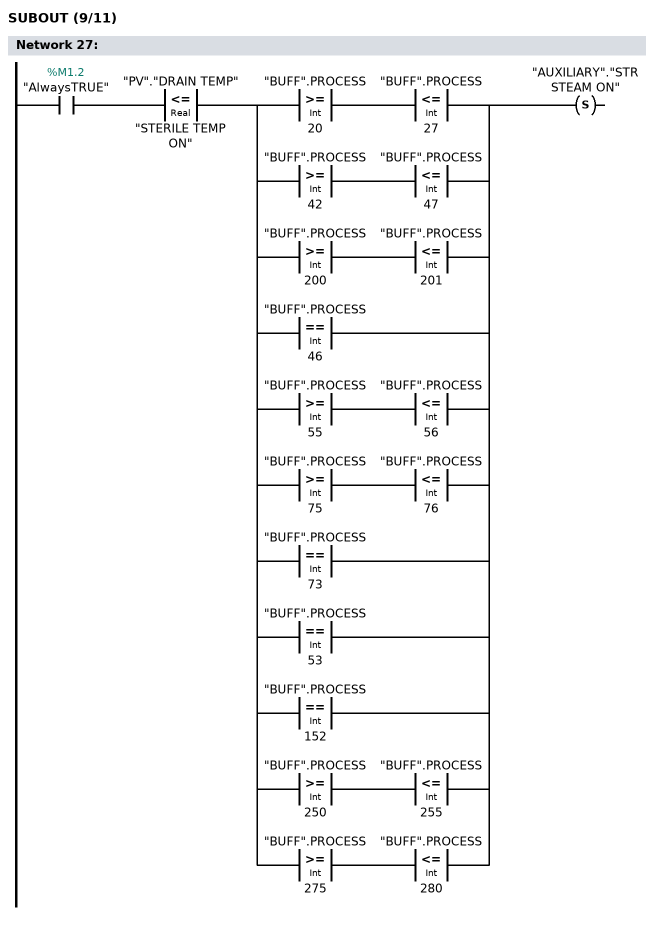
   RUNG wire#powerrail
      Contact( "AlwaysTRUE" )
      { S7_Templates := "SrcType := Real" } LE_Contact(in1 := "PV"."DRAIN TEMP", in2 := "STERILE TEMP ON")
      wire#w1
      { S7_Templates := "SrcType := Int" } GE_Contact(in1 := "BUFF".PROCESS, in2 := 20)
      { S7_Templates := "SrcType := Int" } LE_Contact(in1 := "BUFF".PROCESS, in2 := 27)
      wire#w2
      S_Coil( "AUXILIARY"."STR STEAM ON" )
   END_RUNG
   RUNG wire#w1
      { S7_Templates := "SrcType := Int" } GE_Contact(in1 := "BUFF".PROCESS, in2 := 42)
      { S7_Templates := "SrcType := Int" } LE_Contact(in1 := "BUFF".PROCESS, in2 := 47)
   END_RUNG wire#w2
   RUNG wire#w1
      { S7_Templates := "SrcType := Int" } GE_Contact(in1 := "BUFF".PROCESS, in2 := 200)
      { S7_Templates := "SrcType := Int" } LE_Contact(in1 := "BUFF".PROCESS, in2 := 201)
   END_RUNG wire#w2
   RUNG wire#w1
      { S7_Templates := "SrcType := Int" } EQ_Contact(in1 := "BUFF".PROCESS, in2 := 46)
   END_RUNG wire#w2
   RUNG wire#w1
      { S7_Templates := "SrcType := Int" } GE_Contact(in1 := "BUFF".PROCESS, in2 := 55)
      { S7_Templates := "SrcType := Int" } LE_Contact(in1 := "BUFF".PROCESS, in2 := 56)
   END_RUNG wire#w2
   RUNG wire#w1
      { S7_Templates := "SrcType := Int" } GE_Contact(in1 := "BUFF".PROCESS, in2 := 75)
      { S7_Templates := "SrcType := Int" } LE_Contact(in1 := "BUFF".PROCESS, in2 := 76)
   END_RUNG wire#w2
   RUNG wire#w1
      { S7_Templates := "SrcType := Int" } EQ_Contact(in1 := "BUFF".PROCESS, in2 := 73)
   END_RUNG wire#w2
   RUNG wire#w1
      { S7_Templates := "SrcType := Int" } EQ_Contact(in1 := "BUFF".PROCESS, in2 := 53)
   END_RUNG wire#w2
   RUNG wire#w1
      { S7_Templates := "SrcType := Int" } EQ_Contact(in1 := "BUFF".PROCESS, in2 := 152)
   END_RUNG wire#w2
   RUNG wire#w1
      { S7_Templates := "SrcType := Int" } GE_Contact(in1 := "BUFF".PROCESS, in2 := 250)
      { S7_Templates := "SrcType := Int" } LE_Contact(in1 := "BUFF".PROCESS, in2 := 255)
   END_RUNG wire#w2
   RUNG wire#w1
      { S7_Templates := "SrcType := Int" } GE_Contact(in1 := "BUFF".PROCESS, in2 := 275)
      { S7_Templates := "SrcType := Int" } LE_Contact(in1 := "BUFF".PROCESS, in2 := 280)
   END_RUNG wire#w2
   // the same network as SCL:
   IF "AlwaysTRUE" AND ("PV"."DRAIN TEMP" <= "STERILE TEMP ON") AND ((("BUFF".PROCESS >= 20) AND ("BUFF".PROCESS <= 27)) OR (("BUFF".PROCESS >= 42) AND ("BUFF".PROCESS <= 47)) OR (("BUFF".PROCESS >= 200) AND ("BUFF".PROCESS <= 201)) OR ("BUFF".PROCESS = 46) OR (("BUFF".PROCESS >= 55) AND ("BUFF".PROCESS <= 56)) OR (("BUFF".PROCESS >= 75) AND ("BUFF".PROCESS <= 76)) OR ("BUFF".PROCESS = 73) OR ("BUFF".PROCESS = 53) OR ("BUFF".PROCESS = 152) OR (("BUFF".PROCESS >= 250) AND ("BUFF".PROCESS <= 255)) OR (("BUFF".PROCESS >= 275) AND ("BUFF".PROCESS <= 280))) THEN
       "AUXILIARY"."STR STEAM ON" := TRUE;
   END_IF;
END_REGION

REGION Network 28
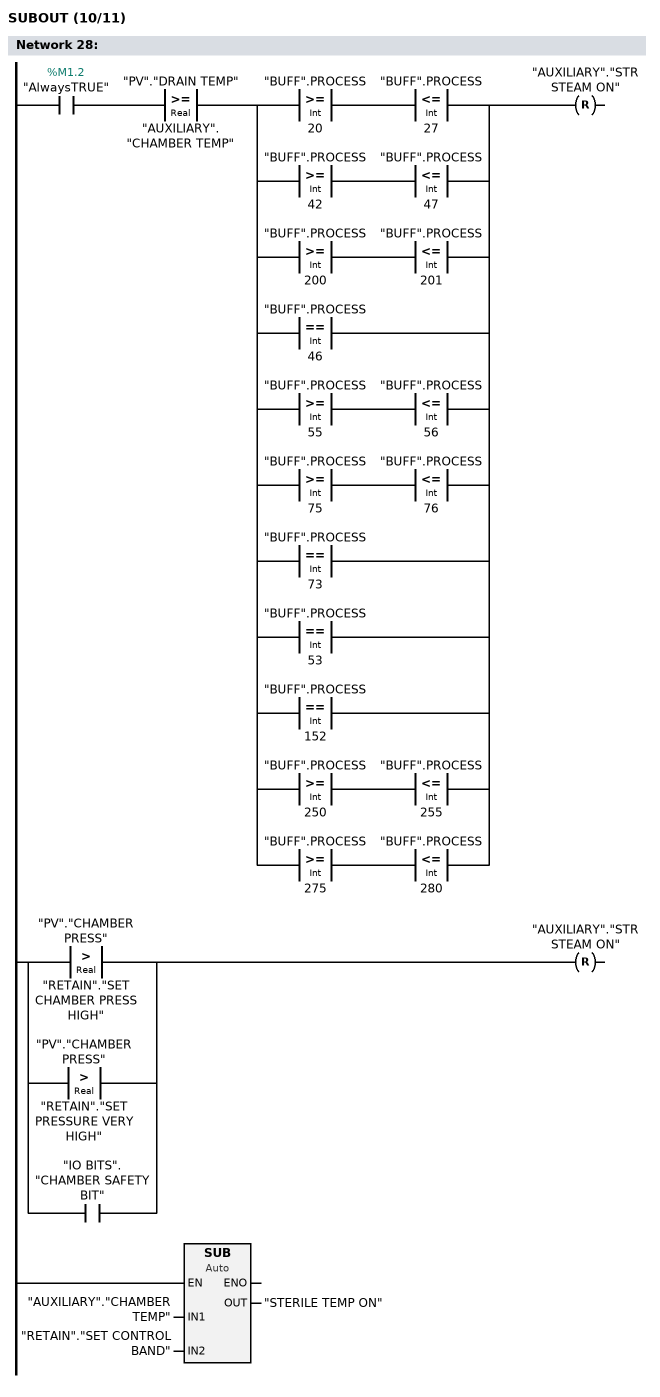
   RUNG wire#powerrail
      Contact( "AlwaysTRUE" )
      { S7_Templates := "SrcType := Real" } GE_Contact(in1 := "PV"."DRAIN TEMP", in2 := "AUXILIARY"."CHAMBER TEMP")
      wire#w1
      { S7_Templates := "SrcType := Int" } GE_Contact(in1 := "BUFF".PROCESS, in2 := 20)
      { S7_Templates := "SrcType := Int" } LE_Contact(in1 := "BUFF".PROCESS, in2 := 27)
      wire#w2
      R_Coil( "AUXILIARY"."STR STEAM ON" )
   END_RUNG
   RUNG wire#w1
      { S7_Templates := "SrcType := Int" } GE_Contact(in1 := "BUFF".PROCESS, in2 := 42)
      { S7_Templates := "SrcType := Int" } LE_Contact(in1 := "BUFF".PROCESS, in2 := 47)
   END_RUNG wire#w2
   RUNG wire#w1
      { S7_Templates := "SrcType := Int" } GE_Contact(in1 := "BUFF".PROCESS, in2 := 200)
      { S7_Templates := "SrcType := Int" } LE_Contact(in1 := "BUFF".PROCESS, in2 := 201)
   END_RUNG wire#w2
   RUNG wire#w1
      { S7_Templates := "SrcType := Int" } EQ_Contact(in1 := "BUFF".PROCESS, in2 := 46)
   END_RUNG wire#w2
   RUNG wire#w1
      { S7_Templates := "SrcType := Int" } GE_Contact(in1 := "BUFF".PROCESS, in2 := 55)
      { S7_Templates := "SrcType := Int" } LE_Contact(in1 := "BUFF".PROCESS, in2 := 56)
   END_RUNG wire#w2
   RUNG wire#w1
      { S7_Templates := "SrcType := Int" } GE_Contact(in1 := "BUFF".PROCESS, in2 := 75)
      { S7_Templates := "SrcType := Int" } LE_Contact(in1 := "BUFF".PROCESS, in2 := 76)
   END_RUNG wire#w2
   RUNG wire#w1
      { S7_Templates := "SrcType := Int" } EQ_Contact(in1 := "BUFF".PROCESS, in2 := 73)
   END_RUNG wire#w2
   RUNG wire#w1
      { S7_Templates := "SrcType := Int" } EQ_Contact(in1 := "BUFF".PROCESS, in2 := 53)
   END_RUNG wire#w2
   RUNG wire#w1
      { S7_Templates := "SrcType := Int" } EQ_Contact(in1 := "BUFF".PROCESS, in2 := 152)
   END_RUNG wire#w2
   RUNG wire#w1
      { S7_Templates := "SrcType := Int" } GE_Contact(in1 := "BUFF".PROCESS, in2 := 250)
      { S7_Templates := "SrcType := Int" } LE_Contact(in1 := "BUFF".PROCESS, in2 := 255)
   END_RUNG wire#w2
   RUNG wire#w1
      { S7_Templates := "SrcType := Int" } GE_Contact(in1 := "BUFF".PROCESS, in2 := 275)
      { S7_Templates := "SrcType := Int" } LE_Contact(in1 := "BUFF".PROCESS, in2 := 280)
   END_RUNG wire#w2
   RUNG wire#powerrail
      { S7_Templates := "SrcType := Real" } GT_Contact(in1 := "PV"."CHAMBER PRESS", in2 := "RETAIN"."SET CHAMBER PRESS HIGH")
      wire#w3
      R_Coil( "AUXILIARY"."STR STEAM ON" )
   END_RUNG
   RUNG wire#powerrail
      { S7_Templates := "SrcType := Real" } GT_Contact(in1 := "PV"."CHAMBER PRESS", in2 := "RETAIN"."SET PRESSURE VERY HIGH")
   END_RUNG wire#w3
   RUNG wire#powerrail
      Contact( "IO BITS"."CHAMBER SAFETY BIT" )
   END_RUNG wire#w3
   RUNG wire#powerrail
      Sub(in1 := "AUXILIARY"."CHAMBER TEMP", in2 := "RETAIN"."SET CONTROL BAND", out => "STERILE TEMP ON")
   END_RUNG
   // the same network as SCL:
   IF "AlwaysTRUE" AND ("PV"."DRAIN TEMP" >= "AUXILIARY"."CHAMBER TEMP") AND ((("BUFF".PROCESS >= 20) AND ("BUFF".PROCESS <= 27)) OR (("BUFF".PROCESS >= 42) AND ("BUFF".PROCESS <= 47)) OR (("BUFF".PROCESS >= 200) AND ("BUFF".PROCESS <= 201)) OR ("BUFF".PROCESS = 46) OR (("BUFF".PROCESS >= 55) AND ("BUFF".PROCESS <= 56)) OR (("BUFF".PROCESS >= 75) AND ("BUFF".PROCESS <= 76)) OR ("BUFF".PROCESS = 73) OR ("BUFF".PROCESS = 53) OR ("BUFF".PROCESS = 152) OR (("BUFF".PROCESS >= 250) AND ("BUFF".PROCESS <= 255)) OR (("BUFF".PROCESS >= 275) AND ("BUFF".PROCESS <= 280))) THEN
       "AUXILIARY"."STR STEAM ON" := FALSE;
   END_IF;
   IF ("PV"."CHAMBER PRESS" > "RETAIN"."SET CHAMBER PRESS HIGH") OR ("PV"."CHAMBER PRESS" > "RETAIN"."SET PRESSURE VERY HIGH") OR "IO BITS"."CHAMBER SAFETY BIT" THEN
       "AUXILIARY"."STR STEAM ON" := FALSE;
   END_IF;
   "STERILE TEMP ON" := "AUXILIARY"."CHAMBER TEMP" - "RETAIN"."SET CONTROL BAND";
END_REGION

REGION Network 29
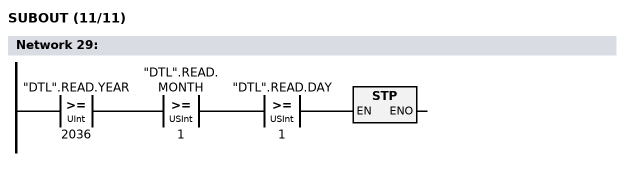
   RUNG wire#powerrail
      { S7_Templates := "SrcType := UInt" } GE_Contact(in1 := "DTL".READ.YEAR, in2 := 2036)
      { S7_Templates := "SrcType := USInt" } GE_Contact(in1 := "DTL".READ.MONTH, in2 := 1)
      { S7_Templates := "SrcType := USInt" } GE_Contact(in1 := "DTL".READ.DAY, in2 := 1)
      STP()
   END_RUNG
   // the same network as SCL:
   IF ("DTL".READ.YEAR >= 2036) AND ("DTL".READ.MONTH >= 1) AND ("DTL".READ.DAY >= 1) THEN STP(); END_IF;
END_REGION
END_FUNCTION

FUNCTION "ZERO L" : Void   // FC10, LAD
{ S7_Optimized_Access := 'TRUE' }
// stored: SetENOAutomatically false
   VAR_TEMP
      "print ok" : String;
   END_VAR
   VAR_TEMP   // added for the SCL form of the ladder/FBD networks
      _w1 : Bool;
      _w2 : Bool;
      _w3 : Bool;
      _w4 : Bool;
      _w5 : Bool;
      _w6 : Bool;
      _w7 : Bool;
      _w8 : Bool;
      _w9 : Bool;
      _w10 : Bool;
      _w11 : Bool;
      _w12 : Bool;
   END_VAR
BEGIN

REGION Network 1
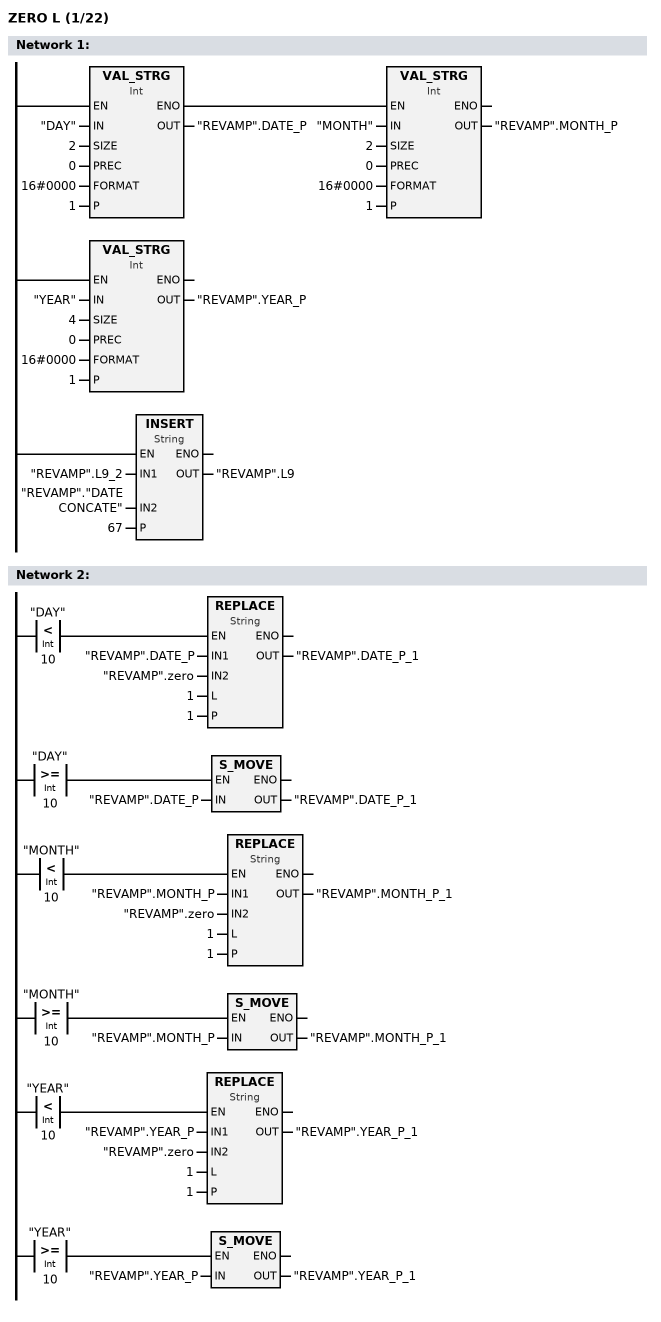
   RUNG wire#powerrail
      { S7_Templates := "[value_type := Int, str_type := String]" } VAL_STRG(IN := "DAY", SIZE := 2, PREC := 0, FORMAT := 16#0000, P := 1, OUT => "REVAMP".DATE_P)
      { S7_Templates := "[value_type := Int, str_type := String]" } VAL_STRG(IN := "MONTH", SIZE := 2, PREC := 0, FORMAT := 16#0000, P := 1, OUT => "REVAMP".MONTH_P)
   END_RUNG
   RUNG wire#powerrail
      { S7_Templates := "[value_type := Int, str_type := String]" } VAL_STRG(IN := "YEAR", SIZE := 4, PREC := 0, FORMAT := 16#0000, P := 1, OUT => "REVAMP".YEAR_P)
   END_RUNG
   RUNG wire#powerrail
      { S7_Templates := "str_type := String" } INSERT(IN1 := "REVAMP".L9_2, IN2 := "REVAMP"."DATE CONCATE", P := 67, OUT => "REVAMP".L9)
   END_RUNG
   // the same network as SCL:
   VAL_STRG(IN := "DAY", SIZE := 2, PREC := 0, FORMAT := 16#0000, P := 1, OUT => "REVAMP".DATE_P, ENO => #_w1);
   IF #_w1 THEN
       VAL_STRG(IN := "MONTH", SIZE := 2, PREC := 0, FORMAT := 16#0000, P := 1, OUT => "REVAMP".MONTH_P);
   END_IF;
   VAL_STRG(IN := "YEAR", SIZE := 4, PREC := 0, FORMAT := 16#0000, P := 1, OUT => "REVAMP".YEAR_P);
   INSERT(IN1 := "REVAMP".L9_2, IN2 := "REVAMP"."DATE CONCATE", P := 67, OUT => "REVAMP".L9);
END_REGION

REGION Network 2
   RUNG wire#powerrail
      { S7_Templates := "SrcType := Int" } LT_Contact(in1 := "DAY", in2 := 10)
      { S7_Templates := "str_type := String" } REPLACE(IN1 := "REVAMP".DATE_P, IN2 := "REVAMP".zero, L := 1, P := 1, OUT => "REVAMP".DATE_P_1)
   END_RUNG
   RUNG wire#powerrail
      { S7_Templates := "SrcType := Int" } GE_Contact(in1 := "DAY", in2 := 10)
      S_Move(in := "REVAMP".DATE_P, out => "REVAMP".DATE_P_1)
   END_RUNG
   RUNG wire#powerrail
      { S7_Templates := "SrcType := Int" } LT_Contact(in1 := "MONTH", in2 := 10)
      { S7_Templates := "str_type := String" } REPLACE(IN1 := "REVAMP".MONTH_P, IN2 := "REVAMP".zero, L := 1, P := 1, OUT => "REVAMP".MONTH_P_1)
   END_RUNG
   RUNG wire#powerrail
      { S7_Templates := "SrcType := Int" } GE_Contact(in1 := "MONTH", in2 := 10)
      S_Move(in := "REVAMP".MONTH_P, out => "REVAMP".MONTH_P_1)
   END_RUNG
   RUNG wire#powerrail
      { S7_Templates := "SrcType := Int" } LT_Contact(in1 := "YEAR", in2 := 10)
      { S7_Templates := "str_type := String" } REPLACE(IN1 := "REVAMP".YEAR_P, IN2 := "REVAMP".zero, L := 1, P := 1, OUT => "REVAMP".YEAR_P_1)
   END_RUNG
   RUNG wire#powerrail
      { S7_Templates := "SrcType := Int" } GE_Contact(in1 := "YEAR", in2 := 10)
      S_Move(in := "REVAMP".YEAR_P, out => "REVAMP".YEAR_P_1)
   END_RUNG
   // the same network as SCL:
   IF "DAY" < 10 THEN
       REPLACE(IN1 := "REVAMP".DATE_P, IN2 := "REVAMP".zero, L := 1, P := 1, OUT => "REVAMP".DATE_P_1);
   END_IF;
   IF "DAY" >= 10 THEN "REVAMP".DATE_P_1 := "REVAMP".DATE_P; END_IF;
   IF "MONTH" < 10 THEN
       REPLACE(IN1 := "REVAMP".MONTH_P, IN2 := "REVAMP".zero, L := 1, P := 1, OUT => "REVAMP".MONTH_P_1);
   END_IF;
   IF "MONTH" >= 10 THEN "REVAMP".MONTH_P_1 := "REVAMP".MONTH_P; END_IF;
   IF "YEAR" < 10 THEN
       REPLACE(IN1 := "REVAMP".YEAR_P, IN2 := "REVAMP".zero, L := 1, P := 1, OUT => "REVAMP".YEAR_P_1);
   END_IF;
   IF "YEAR" >= 10 THEN "REVAMP".YEAR_P_1 := "REVAMP".YEAR_P; END_IF;
END_REGION

REGION Network 3
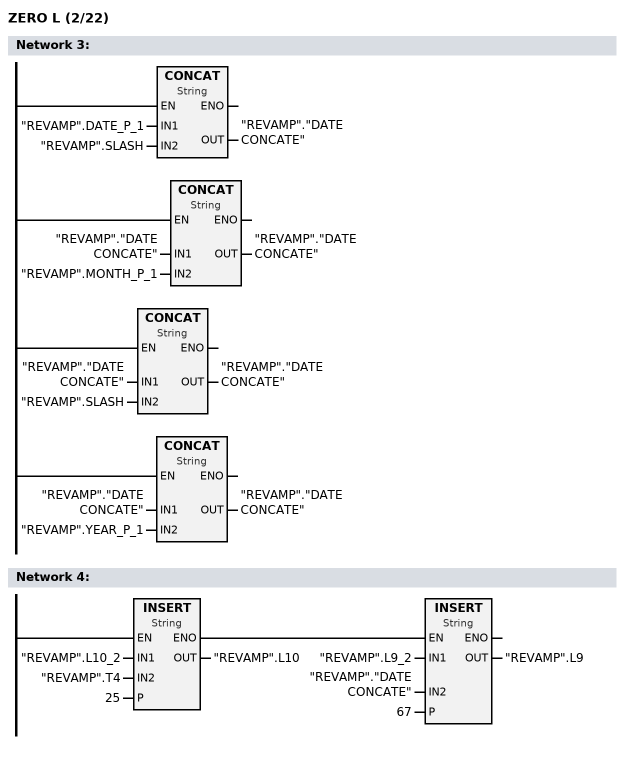
   RUNG wire#powerrail
      { S7_Templates := "[card := 2, str_type := String]" } CONCAT(IN1 := "REVAMP".DATE_P_1, IN2 := "REVAMP".SLASH, OUT => "REVAMP"."DATE CONCATE")
   END_RUNG
   RUNG wire#powerrail
      { S7_Templates := "[card := 2, str_type := String]" } CONCAT(IN1 := "REVAMP"."DATE CONCATE", IN2 := "REVAMP".MONTH_P_1, OUT => "REVAMP"."DATE CONCATE")
   END_RUNG
   RUNG wire#powerrail
      { S7_Templates := "[card := 2, str_type := String]" } CONCAT(IN1 := "REVAMP"."DATE CONCATE", IN2 := "REVAMP".SLASH, OUT => "REVAMP"."DATE CONCATE")
   END_RUNG
   RUNG wire#powerrail
      { S7_Templates := "[card := 2, str_type := String]" } CONCAT(IN1 := "REVAMP"."DATE CONCATE", IN2 := "REVAMP".YEAR_P_1, OUT => "REVAMP"."DATE CONCATE")
   END_RUNG
   // the same network as SCL:
   CONCAT(IN1 := "REVAMP".DATE_P_1, IN2 := "REVAMP".SLASH, OUT => "REVAMP"."DATE CONCATE");
   CONCAT(IN1 := "REVAMP"."DATE CONCATE", IN2 := "REVAMP".MONTH_P_1, OUT => "REVAMP"."DATE CONCATE");
   CONCAT(IN1 := "REVAMP"."DATE CONCATE", IN2 := "REVAMP".SLASH, OUT => "REVAMP"."DATE CONCATE");
   CONCAT(IN1 := "REVAMP"."DATE CONCATE", IN2 := "REVAMP".YEAR_P_1, OUT => "REVAMP"."DATE CONCATE");
END_REGION

REGION Network 4
   RUNG wire#powerrail
      { S7_Templates := "str_type := String" } INSERT(IN1 := "REVAMP".L10_2, IN2 := "REVAMP".T4, P := 25, OUT => "REVAMP".L10)
      { S7_Templates := "str_type := String" } INSERT(IN1 := "REVAMP".L9_2, IN2 := "REVAMP"."DATE CONCATE", P := 67, OUT => "REVAMP".L9)
   END_RUNG
   // the same network as SCL:
   INSERT(IN1 := "REVAMP".L10_2, IN2 := "REVAMP".T4, P := 25, OUT => "REVAMP".L10, ENO => #_w1);
   IF #_w1 THEN
       INSERT(IN1 := "REVAMP".L9_2, IN2 := "REVAMP"."DATE CONCATE", P := 67, OUT => "REVAMP".L9);
   END_IF;
END_REGION

REGION Network 5
